// ---- 20_Product/10_BCF/11_Conv/15_Subsystem/01_DUTs/ST_SubSystemData.TcDUT
TYPE ST_SubsystemData :
(**************************************************************************************
 * 	Application		:	BoxControl Framework
 *	Revision		:	$Revision: 404529 $
 *	Revision date	:	$Date: 2018-04-23 08:21:38 +0200 (Mo., 23 Apr 2018) $
 *	Last changed by	:	$Author: b7bolm $
 *	URL				:	$URL: http://almscdc.swisslog.com/repo/SWPD/Development/BoxControlFramework/20_Release/trunk/01_Software/BCF/BCF/JumpStart/20_Product/10_App/15_Subsystem/10_Lib/10_Conv/01_DUTs/ST_SubSystemData.TcDUT $
 *
 *	Purpose			:	Subsystem data
 *
 * ------------------------------------------------------------------------------------
 *	Copyright Swisslog [IP AG], Switzerland. All rights reserved.
 * 
 * ------------------------------------------------------------------------------------
 *	
 * 	Revision History: 
 *
 * 	VERSION			DATE			INITIALS			DESCRIPTION
 *	0.1				01.01.2001		swl					Example
 *
 **************************************************************************************)
STRUCT
	Init			: BOOL; // Initialized
	InitRunning		: BOOL; // Init ongoing
	OperationState	: ST_PositionState; // Subsystem state
	ErrorData		: ST_SubsystemErrorStruct; // Error data set 
END_STRUCT
END_TYPE

// ---- 20_Product/10_BCF/11_Conv/15_Subsystem/01_DUTs/ST_SubSystemErrorStruct.TcDUT
TYPE ST_SubsystemErrorStruct :
(**************************************************************************************
 * 	Application		:	BoxControl Framework
 *	Revision		:	$Revision: 404529 $
 *	Revision date	:	$Date: 2018-04-23 08:21:38 +0200 (Mo., 23 Apr 2018) $
 *	Last changed by	:	$Author: b7bolm $
 *	URL				:	$URL: http://almscdc.swisslog.com/repo/SWPD/Development/BoxControlFramework/20_Release/trunk/01_Software/BCF/BCF/JumpStart/20_Product/10_App/15_Subsystem/10_Lib/10_Conv/01_DUTs/ST_SubSystemErrorStruct.TcDUT $
 *
 *	Purpose			:	Group error structure - Contains all information for the
 *						error handling.
 *
 * ------------------------------------------------------------------------------------
 *	Copyright Swisslog [IP AG], Switzerland. All rights reserved.
 * 
 * ------------------------------------------------------------------------------------
 *	
 * 	Revision History: 
 *
 * 	VERSION			DATE			INITIALS			DESCRIPTION
 *	0.1				01.01.2001		swl					Example
 *
 **************************************************************************************)
STRUCT
	ErrorState				: E_ErrorState; // Ongoing module error state
	Error					: ST_ErrorDataSet; // Ongoing reported error
	DataSetIdx				: INT; // Choosen error set index
	ErrorDataSet			: ARRAY [1..NUMBER_OF_ERROR_SETS] OF ST_ErrorDataSet; // Overview about all message sets
	ExternalError			: ST_ErrorDataSet; // External error, Can be set customized or by control code
	GroupErrorPending		: BOOL; // A group is in error state
END_STRUCT
END_TYPE

// ---- 20_Product/10_BCF/11_Conv/15_Subsystem/01_DUTs/ST_SubSystemInterface.TcDUT
TYPE ST_SubsystemInterface :
(**************************************************************************************
 * 	Application		:	BoxControl Framework
 *	Revision		:	$Revision: 404529 $
 *	Revision date	:	$Date: 2018-04-23 08:21:38 +0200 (Mo., 23 Apr 2018) $
 *	Last changed by	:	$Author: b7bolm $
 *	URL				:	$URL: http://almscdc.swisslog.com/repo/SWPD/Development/BoxControlFramework/20_Release/trunk/01_Software/BCF/BCF/JumpStart/20_Product/10_App/15_Subsystem/10_Lib/10_Conv/01_DUTs/ST_SubSystemInterface.TcDUT $
 *
 *	Purpose			:	
 *
 * ------------------------------------------------------------------------------------
 *	Copyright Swisslog [IP AG], Switzerland. All rights reserved.
 * 
 * ------------------------------------------------------------------------------------
 *	
 * 	Revision History: 
 *
 * 	VERSION			DATE			INITIALS			DESCRIPTION
 *	0.1				01.01.2001		swl					Example
 *
 **************************************************************************************)
STRUCT
	In			: ST_SubSystemInterfaceIn;
	Out			: ST_SubSystemInterfaceOut;
END_STRUCT
END_TYPE

// ---- 20_Product/10_BCF/11_Conv/15_Subsystem/01_DUTs/ST_SubSystemInterfaceIn.TcDUT
TYPE ST_SubSystemInterfaceIn :
(**************************************************************************************
 * 	Application		:	BoxControl Framework
 *	Revision		:	$Revision: 404529 $
 *	Revision date	:	$Date: 2018-04-23 08:21:38 +0200 (Mo., 23 Apr 2018) $
 *	Last changed by	:	$Author: b7bolm $
 *	URL				:	$URL: http://almscdc.swisslog.com/repo/SWPD/Development/BoxControlFramework/20_Release/trunk/01_Software/BCF/BCF/JumpStart/20_Product/10_App/15_Subsystem/10_Lib/10_Conv/01_DUTs/ST_SubSystemInterfaceIn.TcDUT $
 *
 *	Purpose			:	
 *
 * ------------------------------------------------------------------------------------
 *	Copyright Swisslog [IP AG], Switzerland. All rights reserved.
 * 
 * ------------------------------------------------------------------------------------
 *	
 * 	Revision History: 
 *
 * 	VERSION			DATE			INITIALS			DESCRIPTION
 *	0.1				01.01.2001		swl					Example
 *
 **************************************************************************************)
STRUCT
	MasterSpeed					: INT; // Incoming Master speed request
END_STRUCT
END_TYPE

// ---- 20_Product/10_BCF/11_Conv/15_Subsystem/01_DUTs/ST_SubSystemInterfaceOut.TcDUT
TYPE ST_SubSystemInterfaceOut :
(**************************************************************************************
 * 	Application		:	BoxControl Framework
 *	Revision		:	$Revision: 404529 $
 *	Revision date	:	$Date: 2018-04-23 08:21:38 +0200 (Mo., 23 Apr 2018) $
 *	Last changed by	:	$Author: b7bolm $
 *	URL				:	$URL: http://almscdc.swisslog.com/repo/SWPD/Development/BoxControlFramework/20_Release/trunk/01_Software/BCF/BCF/JumpStart/20_Product/10_App/15_Subsystem/10_Lib/10_Conv/01_DUTs/ST_SubSystemInterfaceOut.TcDUT $
 *
 *	Purpose			:	
 *
 * ------------------------------------------------------------------------------------
 *	Copyright Swisslog [IP AG], Switzerland. All rights reserved.
 * 
 * ------------------------------------------------------------------------------------
 *	
 * 	Revision History: 
 *
 * 	VERSION			DATE			INITIALS			DESCRIPTION
 *	0.1				01.01.2001		swl					Example
 *
 **************************************************************************************)
STRUCT
	MasterSpeed					: INT; // Valid master speed
END_STRUCT
END_TYPE

// ---- 20_Product/20_ProBox/10_Base/01_DUTs/E_ErrorProduct.TcDUT
{attribute 'qualified_only'}
{attribute 'strict'}
(**************************************************************************************
 * 	Application		:	BoxControl Framework
 *	Revision		:	$Revision: 417092 $
 *	Revision date	:	$Date: 2018-11-14 12:58:58 +0100 (Mi., 14 Nov 2018) $
 *	Last changed by	:	$Author: q8aberh $
 *	URL				:	$URL: http://almscdc.swisslog.com/repo/SWPD/Development/ProMove/02_Controls/ProBox/03_Implementation/01_DevelopmentProject/01_Software/ProBox_COE/ProBox_DevProj_v1.0/PLC_1/20_Product/10_App/10_Base/E_ErrorProduct.TcDUT $
 *
 *	Purpose			:	Product error
 *						This Structure can be used for product specific error codes.
 *						ATTENTION! - WM needs to be updated for each error code
 *
 *						0 - 999 Reserved Framework
 *						1000... Product specific
 *
 * ------------------------------------------------------------------------------------
 *	Copyright Swisslog [IP AG], Switzerland. All rights reserved.
 * 
 * ------------------------------------------------------------------------------------
 *	
 * 	Revision History: 
 *
 * 	VERSION			DATE			INITIALS			DESCRIPTION
 *	0.1				01.01.2001		swl					Example
 *
 **************************************************************************************)
TYPE E_ErrorProduct :
(
	UNDEF := 1000,	
(* -------------------------------------------------------------
		ProBox error messages
--------------------------------------------------------------*)
	SCALE_OVER_UNDER_WEIGHT							:= 1100,
	SCALE_WEIGHT_CELL_ERROR							:= 1101
	
);
END_TYPE

// ---- 20_Product/20_ProBox/22_ProMove/01_DUTs/ASI/ST_ASI_HW_Input.TcDUT
TYPE ST_ASI_HW_Input :
STRUCT
	A_1_15              AT %I* : ST_HW_InputsASi_1_15;  //Slave A 1..15
	A_16_31             AT %I* : ST_HW_InputsASi_16_31; //Slave A 16..31
	B_1_15              AT %I* : ST_HW_InputsASi_1_15;  //Slave B 1..15
	B_16_31             AT %I* : ST_HW_InputsASi_16_31; //Slave B 16..31
END_STRUCT
END_TYPE

// ---- 20_Product/20_ProBox/22_ProMove/01_DUTs/ASI/ST_ASI_HW_IO.TcDUT
TYPE ST_ASI_HW_IO :
STRUCT
	I 	AT %I* : ST_ASI_HW_Input; //ASI Ring 1 Inputs
	//I2 : ST_ASI_HW_Input; //ASI Ring 2 Inputs
	Q 	AT %Q* : ST_ASI_HW_Output; //ASI ring 1 Outputs
	//Q2 : ST_ASI_HW_Output; //ASI ring 2 Outputs
END_STRUCT
END_TYPE

// ---- 20_Product/20_ProBox/22_ProMove/01_DUTs/ASI/ST_ASI_HW_Output.TcDUT
TYPE ST_ASI_HW_Output :
STRUCT
	A_1_15              AT %Q* : ST_HW_OutputsASi_1_15;  //Slave A 1..15
	A_16_31             AT %Q* : ST_HW_OutputsASi_16_31; //Slave A 16..31
	B_1_15              AT %Q* : ST_HW_OutputsASi_1_15;  //Slave B 1..15
	B_16_31             AT %Q* : ST_HW_OutputsASi_16_31; //Slave B 16..31
END_STRUCT
END_TYPE

// ---- 20_Product/20_ProBox/22_ProMove/01_DUTs/ASI/ST_HW_InputsASi_16_31.TcDUT
TYPE ST_HW_InputsASi_16_31 :
STRUCT
	IN_17_1	: BIT;
	IN_17_2	: BIT;
	IN_17_3	: BIT;
	IN_17_4 	: BIT;
	
	IN_16_1	: BIT;
	IN_16_2	: BIT;
	IN_16_3	: BIT;
	IN_16_4 	: BIT;

	IN_19_1	: BIT;
	IN_19_2	: BIT;
	IN_19_3	: BIT;
	IN_19_4	: BIT;

	IN_18_1	: BIT;
	IN_18_2	: BIT;
	IN_18_3	: BIT;
	IN_18_4	: BIT;

	IN_21_1	: BIT;
	IN_21_2	: BIT;
	IN_21_3	: BIT;
	IN_21_4 	: BIT;
	
	IN_20_1	: BIT;
	IN_20_2	: BIT;
	IN_20_3	: BIT;
	IN_20_4	: BIT;

	IN_23_1	: BIT;
	IN_23_2	: BIT;
	IN_23_3	: BIT;
	IN_23_4 	: BIT;

	IN_22_1	: BIT;
	IN_22_2	: BIT;
	IN_22_3	: BIT;
	IN_22_4	: BIT;

	IN_25_1	: BIT;
	IN_25_2	: BIT;
	IN_25_3	: BIT;
	IN_25_4	: BIT;

	IN_24_1	: BIT;
	IN_24_2	: BIT;
	IN_24_3	: BIT;
	IN_24_4	: BIT;

	IN_27_1	: BIT;
	IN_27_2	: BIT;
	IN_27_3	: BIT;
	IN_27_4	: BIT;

	IN_26_1	: BIT;
	IN_26_2	: BIT;
	IN_26_3	: BIT;
	IN_26_4	: BIT;

	IN_29_1	: BIT;
	IN_29_2	: BIT;
	IN_29_3	: BIT;
	IN_29_4	: BIT;

	IN_28_1	: BIT;
	IN_28_2	: BIT;
	IN_28_3	: BIT;
	IN_28_4	: BIT;
	
	IN_31_1	: BIT;
	IN_31_2	: BIT;
	IN_31_3	: BIT;
	IN_31_4	: BIT;

	IN_30_1	: BIT;
	IN_30_2	: BIT;
	IN_30_3	: BIT;
	IN_30_4	: BIT;
END_STRUCT
END_TYPE

// ---- 20_Product/20_ProBox/22_ProMove/01_DUTs/ASI/ST_HW_InputsASi_1_15.TcDUT
TYPE ST_HW_InputsASi_1_15 :
STRUCT
	IN_1_1	: BIT;
	IN_1_2	: BIT;
	IN_1_3	: BIT;
	IN_1_4 	: BIT;
	
	CONF_ERR		: BIT;
	ASI_POWER_FAULT	: BIT;
	NODE_ERROR		: BIT;
	CONFIG_MODE		: BIT;

	IN_3_1	: BIT;
	IN_3_2	: BIT;
	IN_3_3	: BIT;
	IN_3_4 	: BIT;

	IN_2_1	: BIT;
	IN_2_2	: BIT;
	IN_2_3	: BIT;
	IN_2_4 	: BIT;

	IN_5_1	: BIT;
	IN_5_2	: BIT;
	IN_5_3	: BIT;
	IN_5_4 	: BIT;
	
	IN_4_1	: BIT;
	IN_4_2	: BIT;
	IN_4_3	: BIT;
	IN_4_4 	: BIT;

	IN_7_1	: BIT;
	IN_7_2	: BIT;
	IN_7_3	: BIT;
	IN_7_4 	: BIT;

	IN_6_1	: BIT;
	IN_6_2	: BIT;
	IN_6_3	: BIT;
	IN_6_4 	: BIT;

	IN_9_1	: BIT;
	IN_9_2	: BIT;
	IN_9_3	: BIT;
	IN_9_4 	: BIT;

	IN_8_1	: BIT;
	IN_8_2	: BIT;
	IN_8_3	: BIT;
	IN_8_4 	: BIT;

	IN_11_1	: BIT;
	IN_11_2	: BIT;
	IN_11_3	: BIT;
	IN_11_4	: BIT;

	IN_10_1	: BIT;
	IN_10_2	: BIT;
	IN_10_3	: BIT;
	IN_10_4	: BIT;

	IN_13_1	: BIT;
	IN_13_2	: BIT;
	IN_13_3	: BIT;
	IN_13_4	: BIT;

	IN_12_1	: BIT;
	IN_12_2	: BIT;
	IN_12_3	: BIT;
	IN_12_4	: BIT;
	
	IN_15_1	: BIT;
	IN_15_2	: BIT;
	IN_15_3	: BIT;
	IN_15_4	: BIT;

	IN_14_1	: BIT;
	IN_14_2	: BIT;
	IN_14_3	: BIT;
	IN_14_4	: BIT;
END_STRUCT
END_TYPE

// ---- 20_Product/20_ProBox/22_ProMove/01_DUTs/ASI/ST_HW_OutputsASi_16_31.TcDUT
TYPE ST_HW_OutputsASi_16_31 :
STRUCT
	OUT_17_1	: BIT;
	OUT_17_2	: BIT;
	OUT_17_3	: BIT;
	OUT_17_4 	: BIT;
	
	OUT_16_1	: BIT;
	OUT_16_2	: BIT;
	OUT_16_3	: BIT;
	OUT_16_4 	: BIT;

	OUT_19_1	: BIT;
	OUT_19_2	: BIT;
	OUT_19_3	: BIT;
	OUT_19_4	: BIT;

	OUT_18_1	: BIT;
	OUT_18_2	: BIT;
	OUT_18_3	: BIT;
	OUT_18_4	: BIT;

	OUT_21_1	: BIT;
	OUT_21_2	: BIT;
	OUT_21_3	: BIT;
	OUT_21_4 	: BIT;
	
	OUT_20_1	: BIT;
	OUT_20_2	: BIT;
	OUT_20_3	: BIT;
	OUT_20_4	: BIT;

	OUT_23_1	: BIT;
	OUT_23_2	: BIT;
	OUT_23_3	: BIT;
	OUT_23_4 	: BIT;

	OUT_22_1	: BIT;
	OUT_22_2	: BIT;
	OUT_22_3	: BIT;
	OUT_22_4	: BIT;

	OUT_25_1	: BIT;
	OUT_25_2	: BIT;
	OUT_25_3	: BIT;
	OUT_25_4	: BIT;

	OUT_24_1	: BIT;
	OUT_24_2	: BIT;
	OUT_24_3	: BIT;
	OUT_24_4	: BIT;

	OUT_27_1	: BIT;
	OUT_27_2	: BIT;
	OUT_27_3	: BIT;
	OUT_27_4	: BIT;

	OUT_26_1	: BIT;
	OUT_26_2	: BIT;
	OUT_26_3	: BIT;
	OUT_26_4	: BIT;

	OUT_29_1	: BIT;
	OUT_29_2	: BIT;
	OUT_29_3	: BIT;
	OUT_29_4	: BIT;

	OUT_28_1	: BIT;
	OUT_28_2	: BIT;
	OUT_28_3	: BIT;
	OUT_28_4	: BIT;
	
	OUT_31_1	: BIT;
	OUT_31_2	: BIT;
	OUT_31_3	: BIT;
	OUT_31_4	: BIT;

	OUT_30_1	: BIT;
	OUT_30_2	: BIT;
	OUT_30_3	: BIT;
	OUT_30_4	: BIT;
END_STRUCT
END_TYPE

// ---- 20_Product/20_ProBox/22_ProMove/01_DUTs/ASI/ST_HW_OutputsASi_1_15.TcDUT
TYPE ST_HW_OutputsASi_1_15 :
STRUCT
	OUT_1_1	: BIT;
	OUT_1_2	: BIT;
	OUT_1_3	: BIT;
	OUT_1_4 : BIT;
	
	SET_OFFLINE			: BIT;
	LOS_MASTER_BIT		: BIT;
	SET_CONFIG_MODE		: BIT;
	SET_PROTECTED_MODE	: BIT;

	OUT_3_1	: BIT;
	OUT_3_2	: BIT;
	OUT_3_3	: BIT;
	OUT_3_4 : BIT;

	OUT_2_1	: BIT;
	OUT_2_2	: BIT;
	OUT_2_3	: BIT;
	OUT_2_4 : BIT;

	OUT_5_1	: BIT;
	OUT_5_2	: BIT;
	OUT_5_3	: BIT;
	OUT_5_4 : BIT;
	
	OUT_4_1	: BIT;
	OUT_4_2	: BIT;
	OUT_4_3	: BIT;
	OUT_4_4 : BIT;

	OUT_7_1	: BIT;
	OUT_7_2	: BIT;
	OUT_7_3	: BIT;
	OUT_7_4 : BIT;

	OUT_6_1	: BIT;
	OUT_6_2	: BIT;
	OUT_6_3	: BIT;
	OUT_6_4 : BIT;

	OUT_9_1	: BIT;
	OUT_9_2	: BIT;
	OUT_9_3	: BIT;
	OUT_9_4 : BIT;

	OUT_8_1	: BIT;
	OUT_8_2	: BIT;
	OUT_8_3	: BIT;
	OUT_8_4 : BIT;

	OUT_11_1	: BIT;
	OUT_11_2	: BIT;
	OUT_11_3	: BIT;
	OUT_11_4	: BIT;

	OUT_10_1	: BIT;
	OUT_10_2	: BIT;
	OUT_10_3	: BIT;
	OUT_10_4	: BIT;

	OUT_13_1	: BIT;
	OUT_13_2	: BIT;
	OUT_13_3	: BIT;
	OUT_13_4	: BIT;

	OUT_12_1	: BIT;
	OUT_12_2	: BIT;
	OUT_12_3	: BIT;
	OUT_12_4	: BIT;
	
	OUT_15_1	: BIT;
	OUT_15_2	: BIT;
	OUT_15_3	: BIT;
	OUT_15_4	: BIT;

	OUT_14_1	: BIT;
	OUT_14_2	: BIT;
	OUT_14_3	: BIT;
	OUT_14_4	: BIT;
END_STRUCT
END_TYPE

// ---- 20_Product/20_ProBox/22_ProMove/01_DUTs/E_Axis_Orientation.TcDUT
TYPE E_Axis_Orientation :
(**************************************************************************************
 * 	Application		:	BoxControl Framework
 *	Revision		:	$Revision: 417092 $
 *	Revision date	:	$Date: 2018-11-14 12:58:58 +0100 (Mi., 14 Nov 2018) $
 *	Last changed by	:	$Author: q8aberh $
 *	URL				:	$URL: http://almscdc.swisslog.com/repo/SWPD/Development/ProMove/02_Controls/ProBox/03_Implementation/01_DevelopmentProject/01_Software/ProBox_COE/ProBox_DevProj_v1.0/PLC_1/20_Product/10_App/12_E_Functions/11_ProBox/01_DUTs/E_Axis_Orientation.TcDUT $
 *
 *	Purpose			:	orientation of function axis on element 
 *
 * ------------------------------------------------------------------------------------
 *	Copyright Swisslog [IP AG], Switzerland. All rights reserved.
 * 
 * ------------------------------------------------------------------------------------
 *	
 * 	Revision History: 
 *
 * 	VERSION			DATE			INITIALS			DESCRIPTION
 *	0.1				15.06.2018		lca					Example
 *
 **************************************************************************************)	
(
	IDLE, // Funciton axis is not requested by an element
	Element_12, // Funciton axis is requested by the element axis 1-2 in the same direction
	Element_21, // Funciton axis is requested by the element axis 1-2 in the opposite direction
	Element_34, // Funciton axis is requested by the element axis 3-4 in the same direction
	Element_43  // Funciton axis is requested by the element axis 3-4 in the opposite direction	
);
END_TYPE

// ---- 20_Product/20_ProBox/22_ProMove/01_DUTs/E_ProBoxMotorSpeed.TcDUT
TYPE E_ProBoxMotorSpeed :
(**************************************************************************************
 * 	Application		:	BoxControl Framework
 *	Revision		:	$Revision: 418851 $
 *	Revision date	:	$Date: 2018-12-11 17:28:45 +0100 (Di., 11 Dez 2018) $
 *	Last changed by	:	$Author: Q8OTTOC $
 *	URL				:	$URL: http://almscdc.swisslog.com/repo/SWPD/Development/ProMove/02_Controls/ProBox/03_Implementation/01_DevelopmentProject/01_Software/ProBox_COE/ProBox_DevProj_v1.0/PLC_1/20_Product/10_App/12_E_Functions/11_ProBox/01_DUTs/E_ProBoxMotorSpeed.TcDUT $
 *
 *	Purpose			:	Motor speed
 *
 * ------------------------------------------------------------------------------------
 *	Copyright Swisslog [IP AG], Switzerland. All rights reserved.
 * 
 * ------------------------------------------------------------------------------------
 *	
 * 	Revision History: 
 *
 * 	VERSION			DATE			INITIALS			DESCRIPTION
 *	0.1				13.04.2018		PkF					First version of motor speeds
  *	0.2				29.11.2018		lca					Sorted from lowest to highest speed
 *
 **************************************************************************************)
(
	CREEP_SPEED,
	LOW_SPEED,
	NORMAL	
);
END_TYPE

// ---- 20_Product/20_ProBox/22_ProMove/15_SubSystem/01_DUTs/ST_CFG_ProBoxSubsystem.TcDUT
TYPE ST_CFG_ProBoxSubsystem :
STRUCT
	AM_Exists					: BOOL; // Automation manager is existing
	SPOC_Exists					: BOOL; // SPOC exists			
	tRequestReset				: TIME; // Time to reset a request
	tDelayMonitoring			: TIME; // Time to delay monitoring	
	tDelayStopping				: TIME; // Time to delay stopping
	EnableTimeSync				: BOOL; // Enable time sync
	MinTimeSync					: TIME; // Minimal time sync value
	CPU_FanExists				: BOOL; // Is true if CPU with fan equiped 
	MinFanSpeed					: UINT; // Min FAN speed
	CPU_UsageWarning			: INT; // CPU usage warning [%]
	CPU_UsageError				: INT; // CPU usage error [%]
	CPU_TemperatureWarning		: INT; // CPU temperatur warning
	CPU_TemperatureError		: INT; // CPU temperatur error
END_STRUCT
END_TYPE

// ---- 20_Product/20_ProBox/30_Toolbox/12_DUTs/E_PalletOrientation.TcDUT
TYPE E_PalletOrientation :
(
	OrientationZero,
	OrientationNinty,
	OrientationOneEighty,
	OrientationTwoSeventy
);
END_TYPE

// ---- 20_Product/20_ProBox/30_Toolbox/70_Strategies/01_DUTs/ST_FifoBuffer.TcDUT
TYPE ST_FifoBuffer :
STRUCT
	Occupied 			: BOOL;
	EntryOK 			: BOOL;
	eFunctionNumber		: E_FunctionNumber;
	Priority 			: INT;
	//TU_Indexs			: ARRAY [1..NUMBER_OF_ZONES_PER_FUNCTION] OF DINT;  //store the TU index for all zones	
END_STRUCT
END_TYPE

// ---- 20_Product/20_ProBox/30_Toolbox/70_Strategies/01_DUTs/ST_RoutingSluggingData.TcDUT
TYPE ST_RoutingSluggingData :
STRUCT
	FunctionsBehind 		: ARRAY[1..20] OF E_FunctionNumber; // Functions to check before function (back)
	FunctionsInfront		: ARRAY[1..20] OF E_FunctionNumber; // Functions to check after function (forward)
	InvalidDestinations		: ARRAY[1..20] OF E_FunctionNumber; // Destinations of pallets behind that should not be considered slugging with
END_STRUCT
END_TYPE

// ---- 20_Product/20_ProBox/40_TC_Visualization/15_PowerStore/DTUs/ST_AccessPanel.TcDUT
TYPE ST_AccessPanel :
STRUCT
	inputs : ST_AccessPanelInputs;
	outputs : ST_AccessPanelOutputs;
END_STRUCT
END_TYPE

// ---- 20_Product/20_ProBox/40_TC_Visualization/15_PowerStore/DTUs/ST_AccessPanelInputs.TcDUT
TYPE ST_AccessPanelInputs :
STRUCT
	PB_ActivateMainContactor : BOOL; // Pushbutton activate main contactor
	PB_AutoOn : BOOL; // Pushbutton activate automatic mode
	PB_EmergencyStopReset : BOOL; // Pushbutton reset emergency stop
	PB_ErrorReset : BOOL; // Pushbutton reset error
	PB_EmergencyStop : BOOL; // Pushbutton Emergency stop
	SW_EntryRequest : BOOL; // Auto/Entry request switch
END_STRUCT
END_TYPE

// ---- 20_Product/20_ProBox/40_TC_Visualization/15_PowerStore/DTUs/ST_AccessPanelOutputs.TcDUT
TYPE ST_AccessPanelOutputs :
STRUCT
	LED_MainContactorActivated :BOOL; // LED-lamp main contactor is activated
	LED_AutoIsOn : BOOL; // LED-lamp automatic mode is activated
	LED_ClearEnterance : BOOL; // LED-lamp clear to enter
	LED_EmergencyStop : BOOL; // LED-lamp emergency stop
	LED_Error : BOOL; // LED-lamp error
END_STRUCT
END_TYPE

// ---- 20_Product/20_ProBox/40_TC_Visualization/15_PowerStore/DTUs/ST_AKcabinetPanel.TcDUT
TYPE ST_AKcabinetPanel :
STRUCT
	inputs : ST_AKcabinetPanelInputs;
	outputs : ST_AKcabinetPanelOutputs;
END_STRUCT
END_TYPE

// ---- 20_Product/20_ProBox/40_TC_Visualization/15_PowerStore/DTUs/ST_AKcabinetPanelInputs.TcDUT
TYPE ST_AKcabinetPanelInputs :
STRUCT
	PB_ActivateMainContactor : BOOL; // Pushbutton activate main contactor
	PB_MainContactorOff : BOOL; // Pushbutton main contactor off
	PB_AutoOn : BOOL; // Pushbutton activate automatic mode
	PB_EmergencyStopReset : BOOL; // Pushbutton reset emergency stop
	PB_ErrorReset : BOOL; // Pushbutton reset error
	PB_EmergencyStop : BOOL; // Pushbutton Emergency stop
	SW_Auto : BOOL; // Auto/Man keyswitch
	PB_VcUp : BOOL; // Lift up vertical conveyor
	PB_VcDown : BOOL; // Lift down vertical conveyor
	
	PB_VcConvLeft : BOOL; // Vertical conveyor Left
	PB_VcConvRight : BOOL; // Vertical conveyor Right
 	
	SW_EntryRequest : BOOL; // Auto/Entry request switch
	SW_EmergencyDrive : BOOL; // Emergency drive
	
END_STRUCT
END_TYPE

// ---- 20_Product/20_ProBox/40_TC_Visualization/15_PowerStore/DTUs/ST_AKcabinetPanelOutputs.TcDUT
TYPE ST_AKcabinetPanelOutputs :
STRUCT
	LED_MainContactorActivated :BOOL; // LED-lamp main contactor is activated
	LED_AutoIsOn : BOOL; // LED-lamp automatic mode is activated
	LED_ClearEnterance : BOOL; // LED-lamp clear to enter
	LED_EmergencyStop : BOOL; // LED-lamp emergency stop
	LED_Error : BOOL; // LED-lamp error
END_STRUCT
END_TYPE

// ---- 20_Product/20_ProBox/40_TC_Visualization/15_PowerStore/DTUs/ST_TransferPanel.TcDUT
TYPE ST_TransferPanel :
STRUCT
	inputs : ST_TransferPanelInputs;
	outputs : ST_TransferPanelOutputs;
END_STRUCT
END_TYPE

// ---- 20_Product/20_ProBox/40_TC_Visualization/15_PowerStore/DTUs/ST_TransferPanelInputs.TcDUT
TYPE ST_TransferPanelInputs :
STRUCT
	PB_ActivateMainContactor : BOOL; // Pushbutton activate main contactor
	PB_MainContactorOff : BOOL; // Pushbutton main contactor off
	PB_AutoOn : BOOL; // Pushbutton activate automatic mode
	PB_EmergencyStopReset : BOOL; // Pushbutton reset emergency stop
	PB_ErrorReset : BOOL; // Pushbutton reset error
	PB_EmergencyStop : BOOL; // Pushbutton Emergency stop
	SW_Auto : BOOL; // Auto/Man keyswitch
	PB_VcUp : BOOL; // Lift up vertical conveyor
	PB_VcDown : BOOL; // Lift down vertical conveyor
	
	PB_VcConvLeft : BOOL; // Vertical conveyor Left
	PB_VcConvRight : BOOL; // Vertical conveyor Right
 	PB_Conv_1_Left : BOOL; // Conveyor 1 Left
	PB_Conv_1_Right : BOOL; // Conveyor 1 Right
	PB_Conv_2_Left : BOOL; // Conveyor 2 Left
	PB_Conv_2_Right : BOOL; // Conveyor 2 Right
	PB_Conv_3_Left : BOOL; // Conveyor 3 Left
	PB_Conv_3_Right : BOOL; // Conveyor 3 Right
	
	PB_AC_ConvLeft : BOOL; // Aisle carrier conveyor Left
	PB_AC_ConvRight : BOOL; // Aisle carrier conveyor Right
	
END_STRUCT
END_TYPE

// ---- 20_Product/20_ProBox/40_TC_Visualization/15_PowerStore/DTUs/ST_TransferPanelOutputs.TcDUT
TYPE ST_TransferPanelOutputs :
STRUCT
	LED_MainContactorActivated :BOOL; // LED-lamp main contactor is activated
	LED_AutoIsOn : BOOL; // LED-lamp automatic mode is activated
	LED_VcStopped : BOOL; // LED-lamp vertical conveyor stopped
	LED_EmergencyStop : BOOL; // LED-lamp emergency stop
	LED_Error : BOOL; // LED-lamp error
END_STRUCT
END_TYPE

// ---- 20_Product/20_ProBox/40_TC_Visualization/15_PowerStore/DTUs/ST_VC_AccessPanel.TcDUT
TYPE ST_VC_AccessPanel :
STRUCT
	inputs : ST_VC_AccessPanelInputs;
	outputs : ST_VC_AccessPanelOutputs;
END_STRUCT
END_TYPE

// ---- 20_Product/20_ProBox/40_TC_Visualization/15_PowerStore/DTUs/ST_VC_AccessPanelInputs.TcDUT
TYPE ST_VC_AccessPanelInputs :
STRUCT
	PB_ActivateMainContactor : BOOL; // Pushbutton activate main contactor
	PB_MainContactorOff : BOOL; // Pushbutton main contactor off
	PB_AutoOn : BOOL; // Pushbutton activate automatic mode
	PB_EmergencyStopReset : BOOL; // Pushbutton reset emergency stop
	PB_ErrorReset : BOOL; // Pushbutton reset error
	PB_EmergencyStop : BOOL; // Pushbutton Emergency stop
	SW_Auto : BOOL; // Auto/Man keyswitch
	PB_VcUp : BOOL; // Lift up vertical conveyor
	PB_VcDown : BOOL; // Lift down vertical conveyor
	
	PB_VcConvLeft : BOOL; // Vertical conveyor Left
	PB_VcConvRight : BOOL; // Vertical conveyor Right
 	
	SW_EntryRequest : BOOL; // Auto/Entry request switch
	SW_EmergencyDrive : BOOL; // Emergency drive
	
END_STRUCT
END_TYPE

// ---- 20_Product/20_ProBox/40_TC_Visualization/15_PowerStore/DTUs/ST_VC_AccessPanelOutputs.TcDUT
TYPE ST_VC_AccessPanelOutputs :
STRUCT
	LED_MainContactorActivated :BOOL; // LED-lamp main contactor is activated
	LED_AutoIsOn : BOOL; // LED-lamp automatic mode is activated
	LED_ClearEnterance : BOOL; // LED-lamp clear to enter
	LED_EmergencyStop : BOOL; // LED-lamp emergency stop
	LED_Error : BOOL; // LED-lamp error
END_STRUCT
END_TYPE

// ---- 20_Product/30_Toolbox/11_Com/10_TCP_Driver/01_DUTs/E_ConnStates.TcDUT
TYPE E_ConnStates :
(**************************************************************************************
 * 	AUTHOR		Swisslog
 * 	LIBRARY		Data types/02_Library/02_Communication/TCP-Driver
 *	RELEASE		1.0.0
 * ------------------------------------------------------------------------------------
 * 	Revision History: 
 *
 * 	VERSION		DATE		INITIALS	DESCRIPTION
 *	0.1		07.09.2011	swl		initial version
 **************************************************************************************)
(
	CONN_IDLE,  // 0
	CONN_RUNNING, // 1
	CONN_CLOSE, // 2
	CONN_ERROR // 3
);
END_TYPE

// ---- 20_Product/30_Toolbox/11_Com/10_TCP_Driver/01_DUTs/E_RecvStates.TcDUT
TYPE E_RecvStates :
(**************************************************************************************
 * 	AUTHOR		Swisslog
 * 	LIBRARY		Data types/02_Library/02_Communication/TCP-Driver
 *	RELEASE		1.0.0
 * ------------------------------------------------------------------------------------
 * 	Revision History: 
 *
 * 	VERSION		DATE		INITIALS	DESCRIPTION
 *	0.1		07.09.2011	swl		initial version
 **************************************************************************************)
(
	RECV_IDLE,
	RECV_WAIT,
	RECV_ERROR
);
END_TYPE

// ---- 20_Product/30_Toolbox/11_Com/10_TCP_Driver/01_DUTs/E_SendStates.TcDUT
TYPE E_SendStates :
(**************************************************************************************
 * 	AUTHOR		Swisslog
 * 	LIBRARY		Data types/02_Library/02_Communication/TCP-Driver
 *	RELEASE		1.0.0
 * ------------------------------------------------------------------------------------
 * 	Revision History: 
 *
 * 	VERSION		DATE		INITIALS	DESCRIPTION
 *	0.1		07.09.2011	swl		initial version
 **************************************************************************************)
(
	SEND_IDLE,
	SEND_WAIT,
	SEND_ERROR
);
END_TYPE

// ---- 20_Product/30_Toolbox/11_Com/10_TCP_Driver/01_DUTs/E_ServStates.TcDUT
TYPE E_ServStates :
(**************************************************************************************
 * 	AUTHOR		Swisslog
 * 	LIBRARY		Data types/02_Library/02_Communication/TCP-Driver
 *	RELEASE		1.0.0
 * ------------------------------------------------------------------------------------
 * 	Revision History: 
 *
 * 	VERSION		DATE		INITIALS	DESCRIPTION
 *	0.1		07.09.2011	swl		initial version
 **************************************************************************************)
(
	ACCEPT_IDLE,
	ACCEPT_OPEN_START,
	ACCEPT_OPEN_WAIT,
	CLIENT_CONNECTED,
	ACCEPT_CLOSE_START,
	ACCEPT_CLOSE_WAIT,
	ACCEPT_ERROR
);
END_TYPE

// ---- 20_Product/30_Toolbox/11_Com/10_TCP_Driver/01_DUTs/ST_CFG_TcpDriver.TcDUT
TYPE ST_CFG_TcpDriver :
(**************************************************************************************
 * 	Application		:	BoxControl Framework
 *	Revision		:	$Revision: 404529 $
 *	Revision date	:	$Date: 2018-04-23 08:21:38 +0200 (Mo., 23 Apr 2018) $
 *	Last changed by	:	$Author: b7bolm $
 *	URL				:	$URL: http://almscdc.swisslog.com/repo/SWPD/Development/BoxControlFramework/20_Release/trunk/01_Software/BCF/BCF/JumpStart/30_Toolbox/11_Com/10_TCP_Driver/01_DUTs/ST_CFG_TcpDriver.TcDUT $
 *
 *	Purpose			:	Configuration TCP/IP channel.
 *
 * ------------------------------------------------------------------------------------
 *	Copyright Swisslog [IP AG], Switzerland. All rights reserved.
 * 
 * ------------------------------------------------------------------------------------
 *	
 * 	Revision History: 
 *
 * 	VERSION			DATE			INITIALS			DESCRIPTION
 *	0.1				01.01.2001		swl					Example
 *
 **************************************************************************************)
STRUCT
	ChannelName				: STRING(80); // Name - Only for debugging
	EnableConnection		: BOOL;	// Enable channel
	RemoteHost				: STRING(15); // IP address of remote host - Client Mode Only! 
	LocalHost				: STRING(15); // IP address of local host - Server Mode Only! 
	RemotePort				: UDINT; // Port of the remote host - Client Mode Only! 
	LocalPort				: UDINT; // Port to listen on - Server Mode Only! 
	Server					: BOOL; // Is this connection to be configured as a server?  (Set to False for Client Mode) 
	ConnectTimeout			: TIME; // Timeout for connection establishment
	ClientRetryInterval		: TIME:= T#45S; // Interval for CLIENT type connections to be re-attempted - default is 45s, RetryInterval should not be lower than 30s to ensure proper execution
	ServerRetryInterval		: TIME:= T#1S; // Interval for SERVER type connections to be re-attempted - default is 1s 
	AcceptPollInterval		: TIME:= T#5S; // Interval for SERVER type connections to poll the port for incoming connection attempts - default is 5s 
	EnableDebugMsg			: BOOL; // Enables sending debug messages	
END_STRUCT
END_TYPE

// ---- 20_Product/30_Toolbox/13_TimerCounter/01_DUTs/E_PulsGen.TcDUT
TYPE E_PulsGen :
(**************************************************************************************
 * 	Application		:	BoxControl Framework
 *	Revision		:	$Revision: 404529 $
 *	Revision date	:	$Date: 2018-04-23 08:21:38 +0200 (Mo., 23 Apr 2018) $
 *	Last changed by	:	$Author: b7bolm $
 *	URL				:	$URL: http://almscdc.swisslog.com/repo/SWPD/Development/BoxControlFramework/20_Release/trunk/01_Software/BCF/BCF/JumpStart/30_Toolbox/13_TimerCounter/01_DUTs/E_PulsGen.TcDUT $
 *
 *	Purpose			:	Pulse generator
 *
 * ------------------------------------------------------------------------------------
 *	Copyright Swisslog [IP AG], Switzerland. All rights reserved.
 * 
 * ------------------------------------------------------------------------------------
 *	
 * 	Revision History: 
 *
 * 	VERSION			DATE			INITIALS			DESCRIPTION
 *	0.1				01.01.2001		swl					Example
 *
 **************************************************************************************)
(
	PG_READY,
	PG_BUSY,
	PG_END
);
END_TYPE

// ---- 20_Product/30_Toolbox/16_Sequencing/01_DUTs/ST_SeqEntry.TcDUT
/// Sequencing data set
TYPE ST_SeqEntry :
(************************************************************************************** 
* 	Application 		: BoxControl Framework 
* 	Revision 			: $Revision: 404877 $ 
* 	Revision date 		: $Date: 2018-04-26 14:10:34 +0200 (Thu, 26 Apr 2018) $ 
* 	Last changed by 	: $Author: b7ernsb $ 
* 	URL 				: $URL: http://almscdc.swisslog.com/repo/SWPD/Development/BoxControlFramework/21_Projects/BCF_2.0/trunk/BCF/BCF/JumpStart/20_Product/10_App/12_E_Functions/10_Lib/10_Conv/FB_FunctionConv.TcPOU $ 
* ------------------------------------------------------------------------------------ 
* 	© Swisslog AG 
* 	Swisslog is not liable for any usage of this source code that is not agreed 
* 	on between Swisslog and the other party. The mandatory legal liability remains 
* 	unaffected. 
* ------------------------------------------------------------------------------------ 
* 	Revision History: 
* 
* 	VERSION 		DATE 			INITIALS 			DESCRIPTION 
* 	0.1 			18.06.2018 		mbo 				Created.
* 
**************************************************************************************)
STRUCT
	TU_Index		: DINT; 
	Sequence		: ULINT; 
	SubSequence		: DINT; 
	TU_ID			: STRING(Conveyor.TU_ID_STRINGLENGTH); 
	TU_ID_HashCode	: ULINT;
	AssignmentID	: UDINT;
	Destination		: ST_PositionIdent;
	DestinationSlot : INT;
	CheckpointID	: STRING(5); 
END_STRUCT
END_TYPE

// ---- 20_Product/30_Toolbox/17_WindowTracking/10_Core/01_DUTs/E_WindowTrackingWindowState.TcDUT
/// Tracking window state
TYPE E_WindowTrackingWindowState :
(************************************************************************************** 
* 	Application 		: BoxControl Framework 
* 	Revision 			: $Revision: 408723 $ 
* 	Revision date 		: $Date: 2018-06-27 13:49:08 +0200 (Wed, 27 Jun 2018) $ 
* 	Last changed by 	: $Author: b7bolm $ 
* 	URL 				: $URL: http://almscdc.swisslog.com/repo/SWPD/Development/BoxControlFramework/21_Projects/BCF_2.0/trunk/BCF/BCF/JumpStart/20_Product/10_App/12_E_Functions/10_Lib/10_Conv/FB_FunctionList.TcPOU $ 
* ------------------------------------------------------------------------------------ 
* 	© Swisslog AG 
* 	Swisslog is not liable for any usage of this source code that is not agreed 
* 	on between Swisslog and the other party. The mandatory legal liability remains 
* 	unaffected. 
* ------------------------------------------------------------------------------------ 
* 	Revision History: 
* 
* 	VERSION 		DATE 			INITIALS 			DESCRIPTION 
* 	0.1 			24.08.2018 		ahe 				First implementation
* 
**************************************************************************************)
(
	IDLE,
	FRONT_EDGE,
	REAR_EDGE,
	OCCUPIED,
	RESERVED
);
END_TYPE

// ---- 20_Product/30_Toolbox/17_WindowTracking/10_Core/01_DUTs/ST_WindowTrackingReloc.TcDUT
TYPE ST_WindowTrackingReloc :
(************************************************************************************** 
* 	Application 		: BoxControl Framework 
* 	Revision 			: $Revision: 408723 $ 
* 	Revision date 		: $Date: 2018-06-27 13:49:08 +0200 (Wed, 27 Jun 2018) $ 
* 	Last changed by 	: $Author: b7bolm $ 
* 	URL 				: $URL: http://almscdc.swisslog.com/repo/SWPD/Development/BoxControlFramework/21_Projects/BCF_2.0/trunk/BCF/BCF/JumpStart/20_Product/10_App/12_E_Functions/10_Lib/10_Conv/FB_FunctionList.TcPOU $ 
* ------------------------------------------------------------------------------------ 
* 	© Swisslog AG 
* 	Swisslog is not liable for any usage of this source code that is not agreed 
* 	on between Swisslog and the other party. The mandatory legal liability remains 
* 	unaffected. 
* ------------------------------------------------------------------------------------ 
* 	Revision History: 
* 
* 	VERSION 		DATE 			INITIALS 			DESCRIPTION 
* 	0.1 			22.08.2018 		herzig 				First implementation
*	0.2				23.08.2018		b7bolm				Review
* 
**************************************************************************************)
STRUCT
	ZoneIndex		: UINT;
	TargetWindow 	: UINT;
END_STRUCT
END_TYPE

// ---- 20_Product/30_Toolbox/17_WindowTracking/10_Core/01_DUTs/ST_WindowTrackingTransfer.TcDUT
TYPE ST_WindowTrackingTransfer :
(**************************************************************************************
 * 	Application		:	BoxControl Framework
 *	Revision		:	$Revision: 351961 $
 *	Revision date	:	$Date: 2015-07-03 16:42:43 +0200 (Fri, 03 Jul 2015) $
 *	Last changed by	:	$Author: d7mangc $
 *	URL				:	$URL: http://almscdc.swisslog.com/repo/SWPD/Development/BoxControlFramework/20_Release/trunk/01_Software/BoxControlFramework/BoxControlFramework/JumpStart/11_Library/10_Application/10_Base/F_CompareAlphaNumericString.TcPOU $
 *
 *	Purpose			:	Window tracking trasnfer data set
 *
 * ------------------------------------------------------------------------------------
 *	Copyright Swisslog [IP AG], Switzerland. All rights reserved.
 * 
 * ------------------------------------------------------------------------------------
 *	
 * 	Revision History: 
 *
 * 	VERSION			DATE			INITIALS			DESCRIPTION
 *	0.1				01.01.2001		swl					Example 
 *
 **************************************************************************************)
STRUCT
	Active					: BOOL;
	AbsoluteInsertPosition	: UDINT;
	ZoneIndex				: UINT;
	LastWindowIndex			: UINT;
END_STRUCT
END_TYPE

// ---- 20_Product/30_Toolbox/17_WindowTracking/10_Core/01_DUTs/ST_WindowTrackingWindow.TcDUT
/// Data of one tracking window
TYPE ST_WindowTrackingWindow :
(************************************************************************************** 
* 	Application 		: BoxControl Framework 
* 	Revision 			: $Revision: 408723 $ 
* 	Revision date 		: $Date: 2018-06-27 13:49:08 +0200 (Wed, 27 Jun 2018) $ 
* 	Last changed by 	: $Author: b7bolm $ 
* 	URL 				: $URL: http://almscdc.swisslog.com/repo/SWPD/Development/BoxControlFramework/21_Projects/BCF_2.0/trunk/BCF/BCF/JumpStart/20_Product/10_App/12_E_Functions/10_Lib/10_Conv/FB_FunctionList.TcPOU $ 
* ------------------------------------------------------------------------------------ 
* 	© Swisslog AG 
* 	Swisslog is not liable for any usage of this source code that is not agreed 
* 	on between Swisslog and the other party. The mandatory legal liability remains 
* 	unaffected. 
* ------------------------------------------------------------------------------------ 
* 	Revision History: 
* 
* 	VERSION 		DATE 			INITIALS 			DESCRIPTION 
* 	0.1 			24.08.2018 		ahe 				First implementation
* 
**************************************************************************************)
STRUCT
	TU_FrontEdgePosition	: UDINT;
	TU_RearEdgePosition		: UDINT;
	State					: E_WindowTrackingWindowState;
	ZoneIndex				: UINT;
	Flush					: BOOL;
END_STRUCT
END_TYPE

// ---- 20_Product/30_Toolbox/17_WindowTracking/10_Core/01_DUTs/ST_WindowTrackingZone.TcDUT
/// Data of one tracking zone
TYPE ST_WindowTrackingZone :
(************************************************************************************** 
* 	Application 		: BoxControl Framework 
* 	Revision 			: $Revision: 408723 $ 
* 	Revision date 		: $Date: 2018-06-27 13:49:08 +0200 (Wed, 27 Jun 2018) $ 
* 	Last changed by 	: $Author: b7bolm $ 
* 	URL 				: $URL: http://almscdc.swisslog.com/repo/SWPD/Development/BoxControlFramework/21_Projects/BCF_2.0/trunk/BCF/BCF/JumpStart/20_Product/10_App/12_E_Functions/10_Lib/10_Conv/FB_FunctionList.TcPOU $ 
* ------------------------------------------------------------------------------------ 
* 	© Swisslog AG 
* 	Swisslog is not liable for any usage of this source code that is not agreed 
* 	on between Swisslog and the other party. The mandatory legal liability remains 
* 	unaffected. 
* ------------------------------------------------------------------------------------ 
* 	Revision History: 
* 
* 	VERSION 		DATE 			INITIALS 			DESCRIPTION 
* 	0.1 			24.08.2018 		ahe 				First implementation
* 
**************************************************************************************)
STRUCT
	Used					: BOOL;
	ActionId				: INT;
	ZoneLength				: UINT;
	ZoneStartWindowIndex	: UINT;
	ZoneEndWindowIndex		: UINT;
	ZoneStartPosition		: UDINT;
	ZoneEndPosition			: UDINT;
	TU_StartWindowIndex		: UINT;
	TU_EndWindowIndex		: UINT;
	TU_Present				: BOOL;
	TU_Index				: DINT;
	Flush					: BOOL; 
	InhibitShifting			: BOOL;
	PositionToLive			: UDINT;
	iActionListener			: I_TrackingActionListener;
END_STRUCT
END_TYPE

// ---- 20_Product/30_Toolbox/17_WindowTracking/10_Core/01_DUTs/ST_ZoneDataPair.TcDUT
TYPE ST_ZoneDataPair :
(************************************************************************************** 
* 	Application 		: BoxControl Framework 
* 	Revision 			: $Revision: 408723 $ 
* 	Revision date 		: $Date: 2018-06-27 13:49:08 +0200 (Wed, 27 Jun 2018) $ 
* 	Last changed by 	: $Author: b7bolm $ 
* 	URL 				: $URL: http://almscdc.swisslog.com/repo/SWPD/Development/BoxControlFramework/21_Projects/BCF_2.0/trunk/BCF/BCF/JumpStart/20_Product/10_App/12_E_Functions/10_Lib/10_Conv/FB_FunctionList.TcPOU $ 
* ------------------------------------------------------------------------------------ 
* 	© Swisslog AG 
* 	Swisslog is not liable for any usage of this source code that is not agreed 
* 	on between Swisslog and the other party. The mandatory legal liability remains 
* 	unaffected. 
* ------------------------------------------------------------------------------------ 
* 	Revision History: 
* 
* 	VERSION 		DATE 			INITIALS 			DESCRIPTION 
* 	0.1 			22.08.2018 		herzig 				First implementation
*	0.2				23.08.2018		b7bolm				Review
* 
**************************************************************************************)
STRUCT
	TrackingZoneIndex	: UINT;
	TU_Index			: DINT;
END_STRUCT
END_TYPE

// ---- 20_Product/30_Toolbox/99_Misc/01_DUTs/E_CPU_InfoStates.TcDUT
{attribute 'qualified_only'}
{attribute 'strict'}
(**************************************************************************************
 * 	Application		:	BoxControl Framework
 *	Revision		:	$Revision: 404529 $
 *	Revision date	:	$Date: 2018-04-23 08:21:38 +0200 (Mo., 23 Apr 2018) $
 *	Last changed by	:	$Author: b7bolm $
 *	URL				:	$URL: http://almscdc.swisslog.com/repo/SWPD/Development/BoxControlFramework/20_Release/trunk/01_Software/BCF/BCF/JumpStart/30_Toolbox/99_Misc/01_DUTs/E_CPU_InfoStates.TcDUT $
 *
 *	Purpose			:	Gathering CPU data
 *
 * ------------------------------------------------------------------------------------
 *	Copyright Swisslog [IP AG], Switzerland. All rights reserved.
 * 
 * ------------------------------------------------------------------------------------
 *	
 * 	Revision History: 
 *
 * 	VERSION			DATE			INITIALS			DESCRIPTION
 *	0.1				01.01.2001		swl					Example
 *
 **************************************************************************************)
TYPE E_CPU_InfoStates :
(
	INIT, 
	READ_DEVICE,
	READ_TEMPERATURE,
	READ_USAGE,
	READ_FAN,
	DONE
);
END_TYPE

// ---- 20_Product/30_Toolbox/99_Misc/13_Helper/01_DUTs/ST_TrackingZoneInfo.TcDUT
TYPE ST_TrackingZoneInfo :
(************************************************************************************** 
* 	Application 		: BoxControl Framework 
* 	Revision 			: $Revision: 408723 $ 
* 	Revision date 		: $Date: 2018-06-27 13:49:08 +0200 (Wed, 27 Jun 2018) $ 
* 	Last changed by 	: $Author: b7bolm $ 
* 	URL 				: $URL: http://almscdc.swisslog.com/repo/SWPD/Development/BoxControlFramework/21_Projects/BCF_2.0/trunk/BCF/BCF/JumpStart/20_Product/10_App/12_E_Functions/10_Lib/10_Conv/FB_FunctionList.TcPOU $ 
* ------------------------------------------------------------------------------------ 
* 	© Swisslog AG 
* 	Swisslog is not liable for any usage of this source code that is not agreed 
* 	on between Swisslog and the other party. The mandatory legal liability remains 
* 	unaffected. 
* ------------------------------------------------------------------------------------ 
* 	Revision History: 
* 
* 	VERSION 		DATE 			INITIALS 			DESCRIPTION 
* 	0.1 			30.11.2018 		mbo					First implementation
* 
**************************************************************************************)
STRUCT
	ZoneIndex		: UINT; // Tracking zone index on tracking
	PositionDelta	: DINT; // Distance to zone start. x < 0 Zone has already passed by x
	ZoneLength		: UINT; // Lengt of tracking zone
END_STRUCT
END_TYPE

// ---- 10_Project/10_App/10_Config/00_GVLs/Groups.TcGVL
///Automatically generated by BoxConfigurator 
VAR_GLOBAL
	fbSG_001                : FB_ProBOXSG;
	fbSG_002                : FB_ProBOXSG;
END_VAR

// ---- 10_Project/10_App/10_Config/00_GVLs/GVL_Safety.TcGVL
///Automatically created by BoxConfigurator
VAR_GLOBAL
END_VAR

// ---- 10_Project/10_App/10_Config/00_GVLs/HardwareMapping.TcGVL
///Automatically created by BoxConfigurator
VAR_GLOBAL
	///ASI HW I/O interface
	AK11_ASI                               : ST_ASI_HW_IO;
	///ASI HW I/O interface
	AK12_ASI                               : ST_ASI_HW_IO;
	///ASI HW I/O interface
	AK13_ASI                               : ST_ASI_HW_IO;
	///Switching group HW interface
	I_10_001_SG                     AT %I* : ST_HW_InputsSG_ProBOX;
	Q_10_001_SG                     AT %Q* : ST_HW_OutputsSG_ProBOX;
	///Switching group HW interface
	I_10_002_SG                     AT %I* : ST_HW_InputsSG_ProBOX;
	Q_10_002_SG                     AT %Q* : ST_HW_OutputsSG_ProBOX;
END_VAR

// ---- 10_Project/10_App/10_Config/00_GVLs/Positions.TcGVL
///Automatically generated by BoxConfigurator 
VAR_GLOBAL
	fbEL_10_001_0200_00_0                   : FB_ProBoxElementMotor;
	fbF_10_001_0200_01_0                    : FB_ProBoxStraightTransport;
	fbF_10_001_0200_02_0                    : FB_InOutFeedAddon;
	fbEL_10_001_0201_00_0                   : FB_ProBoxElementMotor;
	fbF_10_001_0201_01_0                    : FB_LowLiftUnit;
	fbEL_10_001_0202_00_0                   : FB_ProBoxElementMotor;
	fbF_10_001_0202_01_0                    : FB_ProBoxStraightTransport;
	fbEL_10_001_0203_00_0                   : FB_ProBoxElementMotor;
	fbF_10_001_0203_01_0                    : FB_ProBoxStraightTransport;
	fbF_10_001_0203_02_0                    : FB_ProfileCheckAddon;
	fbF_10_001_0203_03_0                    : FB_SickScannerAddon;
	fbF_10_001_0203_04_0                    : FB_TLB4WeightAddon;
	fbF_10_001_0203_05_0                    : FB_PalletCheckAddon;
	fbEL_10_001_0204_00_0                   : FB_ProBoxElementMotor;
	fbF_10_001_0204_01_0                    : FB_TurnTable;
	fbEL_10_001_0205_00_0                   : FB_ProBoxElementMotor;
	fbEL_10_001_0207_00_0                   : FB_ProBoxElementMotor;
	fbF_10_001_0207_01_0                    : FB_ProBoxStraightTransport;
	fbF_10_001_0207_02_0                    : FB_PalletMagazineAddon;
	fbEL_10_001_0208_00_0                   : FB_ProBoxElementMotor;
	fbF_10_001_0208_01_0                    : FB_ProBoxStraightTransport;
	fbEL_10_001_0209_00_0                   : FB_ProBoxElementMotor;
	fbF_10_001_0209_01_0                    : FB_TransferUnit;
	fbEL_10_001_0211_00_0                   : FB_ProBoxElementMotor;
	fbF_10_001_0211_01_0                    : FB_ProBoxStraightTransport;
	fbEL_10_001_0212_00_0                   : FB_ProBoxElementMotor;
	fbF_10_001_0212_01_0                    : FB_TransferUnit;
	fbEL_10_001_0213_00_0                   : FB_ProBoxElementMotor;
	fbF_10_001_0213_01_0                    : FB_ProBoxStraightTransport;
	fbF_10_001_0213_02_0                    : FB_PalletMagazineAddon;
	fbEL_10_001_0214_00_0                   : FB_ProBoxElementMotor;
	fbF_10_001_0214_01_0                    : FB_ProBoxStraightTransport;
	fbEL_10_001_0215_00_0                   : FB_ProBoxElementMotor;
	fbF_10_001_0215_01_0                    : FB_ProBoxStraightTransport;
	fbF_10_001_0215_02_0                    : FB_ProBoxStraightTransport;
	fbF_10_001_0215_03_0                    : FB_CraneXoverAddon;
	fbEL_10_001_0216_00_0                   : FB_ProBoxElementMotor;
	fbF_10_001_0216_01_0                    : FB_ProBoxStraightTransport;
	fbF_10_001_0216_02_0                    : FB_CraneXoverAddon;
	fbEL_10_001_0217_00_0                   : FB_ProBoxElementMotor;
	fbF_10_001_0217_01_0                    : FB_ProBoxStraightTransport;
	fbEL_10_001_0218_00_0                   : FB_ProBoxElementMotor;
	fbF_10_001_0218_01_0                    : FB_ProBoxStraightTransport;
	fbEL_10_001_0219_00_0                   : FB_ProBoxElementMotor;
	fbF_10_001_0219_01_0                    : FB_ProBoxStraightTransport;
	fbEL_10_001_0220_00_0                   : FB_ProBoxElementMotor;
	fbF_10_001_0220_01_0                    : FB_ProBoxStraightTransport;
	fbEL_10_001_0221_00_0                   : FB_ProBoxElementMotor;
	fbF_10_001_0221_01_0                    : FB_TransferUnit;
	fbEL_10_001_0222_00_0                   : FB_ProBoxElementMotor;
	fbF_10_001_0222_01_0                    : FB_TransferUnit;
	fbEL_10_001_0223_00_0                   : FB_ProBoxElementMotor;
	fbEL_10_001_0225_00_0                   : FB_ProBoxElementMotor;
	fbF_10_001_0225_01_0                    : FB_ProBoxStraightTransport;
	fbEL_10_001_0226_00_0                   : FB_ProBoxElementMotor;
	fbF_10_001_0226_01_0                    : FB_ProBoxStraightTransport;
	fbEL_10_001_0227_00_0                   : FB_ProBoxElementMotor;
	fbF_10_001_0227_01_0                    : FB_ProBoxStraightTransport;
	fbEL_10_001_0230_00_0                   : FB_ProBoxElementMotor;
	fbF_10_001_0230_01_0                    : FB_TransferCC;
	fbEL_10_001_0232_00_0                   : FB_ProBoxElementMotor;
	fbF_10_001_0232_01_0                    : FB_ProBoxStraightTransport;
	fbF_10_001_0232_02_0                    : FB_InOutFeedAddon;
	fbEL_10_001_0233_00_0                   : FB_ProBoxElementMotor;
	fbF_10_001_0233_01_0                    : FB_ProBoxStraightTransport;
	fbEL_10_002_0206_00_0                   : FB_ProBoxElementMotor;
	fbF_10_002_0206_01_0                    : FB_ProBoxStraightTransport;
END_VAR

// ---- 10_Project/10_App/10_Config/00_GVLs/ProBoxSystem.TcGVL
///Automatically created by BoxConfigurator
VAR_GLOBAL
	///Set manually to true in order to run Emulation
	EMULATION_ENABLED: BOOL:=TRUE;
	///Set manually to true in when Demo3D emulation is used.
	DEMO3D_SIM_ENABLED: BOOL:=FALSE;
	///Emulation speed. [mm/s]
	EMULATION_SPEED: INT:=1000;
	///SIS_BaseDrive - Time after a message will be repeated (Send)
	REPEAT_TIMEOUT: TIME:=T#10s;
	///SIS_BaseDrive - Time after a DUM telegram is sent
	IDLE_TIMEOUT: TIME:=T#1M;
	///SIS_BaseDrive - Time after connection will be reestablished 
	LINK_LOSS_TIMEOUT: TIME:=T#1M10s;
END_VAR

// ---- 10_Project/10_App/10_Config/00_GVLs/Subsystem.TcGVL
///Automatically created by BoxConfigurator
VAR_GLOBAL
	///Subsystem number 10
	fbSubsystem10: FB_ProBoxSubsystem;
	END_VAR VAR_GLOBAL CONSTANT NUMBERS_OF_ETHERCAT_SLAVE_DIAG: int :=50; //Number of EtherCAT Slaves;
END_VAR

// ---- 10_Project/10_App/12_FlowControl/00_GVLs/FlowControl.TcGVL
///Automatically created by BoxConfigurator
VAR_GLOBAL
	///Main merging service
	fbMergingService: FB_MergingService;
	///Main routing service
	fbRoutingService: FB_RoutingService;
END_VAR

// ---- 10_Project/11_Emu/10_Config/00_GVLs/GroupsEmulation.TcGVL
///Automatically generated by BoxConfigurator 
VAR_GLOBAL
	fbSG_001_Emulation                : FB_ProBOXSG_Emulation;
	fbSG_002_Emulation                : FB_ProBOXSG_Emulation;
END_VAR

// ---- 10_Project/11_Emu/10_Config/00_GVLs/PositionsEmulation.TcGVL
///Automatically generated by BoxConfigurator 
VAR_GLOBAL
	fbEL_10_001_0200_00_0_Emulation         : FB_ProBoxElementMotorEmulation;
	fbF_10_001_0200_01_0_Emulation          : FB_ProBoxStraightTransportEmulation;
	fbF_10_001_0200_02_0_Emulation          : FB_InOutFeedAddonEmulation;
	fbEL_10_001_0201_00_0_Emulation         : FB_ProBoxElementMotorEmulation;
	fbF_10_001_0201_01_0_Emulation          : FB_LowLiftUnitEmulation;
	fbEL_10_001_0202_00_0_Emulation         : FB_ProBoxElementMotorEmulation;
	fbF_10_001_0202_01_0_Emulation          : FB_ProBoxStraightTransportEmulation;
	fbEL_10_001_0203_00_0_Emulation         : FB_ProBoxElementMotorEmulation;
	fbF_10_001_0203_01_0_Emulation          : FB_ProBoxStraightTransportEmulation;
	fbF_10_001_0203_02_0_Emulation          : FB_ProfileCheckAddonEmulation;
	fbF_10_001_0203_03_0_Emulation          : FB_SickScannerAddonEmulation;
	fbF_10_001_0203_04_0_Emulation          : FB_TLB4WeightAddonEmulation;
	fbF_10_001_0203_05_0_Emulation          : FB_PalletCheckAddonEmulation;
	fbEL_10_001_0204_00_0_Emulation         : FB_ProBoxElementMotorEmulation;
	fbF_10_001_0204_01_0_Emulation          : FB_TurnTableEmulation;
	fbEL_10_001_0205_00_0_Emulation         : FB_ProBoxElementMotorEmulation;
	fbEL_10_001_0207_00_0_Emulation         : FB_ProBoxElementMotorEmulation;
	fbF_10_001_0207_01_0_Emulation          : FB_ProBoxStraightTransportEmulation;
	fbF_10_001_0207_02_0_Emulation          : FB_PalletMagazineAddonEmulation;
	fbEL_10_001_0208_00_0_Emulation         : FB_ProBoxElementMotorEmulation;
	fbF_10_001_0208_01_0_Emulation          : FB_ProBoxStraightTransportEmulation;
	fbEL_10_001_0209_00_0_Emulation         : FB_ProBoxElementMotorEmulation;
	fbF_10_001_0209_01_0_Emulation          : FB_TransferUnitEmulation;
	fbEL_10_001_0211_00_0_Emulation         : FB_ProBoxElementMotorEmulation;
	fbF_10_001_0211_01_0_Emulation          : FB_ProBoxStraightTransportEmulation;
	fbEL_10_001_0212_00_0_Emulation         : FB_ProBoxElementMotorEmulation;
	fbF_10_001_0212_01_0_Emulation          : FB_TransferUnitEmulation;
	fbEL_10_001_0213_00_0_Emulation         : FB_ProBoxElementMotorEmulation;
	fbF_10_001_0213_01_0_Emulation          : FB_ProBoxStraightTransportEmulation;
	fbF_10_001_0213_02_0_Emulation          : FB_PalletMagazineAddonEmulation;
	fbEL_10_001_0214_00_0_Emulation         : FB_ProBoxElementMotorEmulation;
	fbF_10_001_0214_01_0_Emulation          : FB_ProBoxStraightTransportEmulation;
	fbEL_10_001_0215_00_0_Emulation         : FB_ProBoxElementMotorEmulation;
	fbF_10_001_0215_01_0_Emulation          : FB_ProBoxStraightTransportEmulation;
	fbF_10_001_0215_02_0_Emulation          : FB_ProBoxStraightTransportEmulation;
	fbF_10_001_0215_03_0_Emulation          : FB_CraneXoverAddonEmulation;
	fbEL_10_001_0216_00_0_Emulation         : FB_ProBoxElementMotorEmulation;
	fbF_10_001_0216_01_0_Emulation          : FB_ProBoxStraightTransportEmulation;
	fbF_10_001_0216_02_0_Emulation          : FB_CraneXoverAddonEmulation;
	fbEL_10_001_0217_00_0_Emulation         : FB_ProBoxElementMotorEmulation;
	fbF_10_001_0217_01_0_Emulation          : FB_ProBoxStraightTransportEmulation;
	fbEL_10_001_0218_00_0_Emulation         : FB_ProBoxElementMotorEmulation;
	fbF_10_001_0218_01_0_Emulation          : FB_ProBoxStraightTransportEmulation;
	fbEL_10_001_0219_00_0_Emulation         : FB_ProBoxElementMotorEmulation;
	fbF_10_001_0219_01_0_Emulation          : FB_ProBoxStraightTransportEmulation;
	fbEL_10_001_0220_00_0_Emulation         : FB_ProBoxElementMotorEmulation;
	fbF_10_001_0220_01_0_Emulation          : FB_ProBoxStraightTransportEmulation;
	fbEL_10_001_0221_00_0_Emulation         : FB_ProBoxElementMotorEmulation;
	fbF_10_001_0221_01_0_Emulation          : FB_TransferUnitEmulation;
	fbEL_10_001_0222_00_0_Emulation         : FB_ProBoxElementMotorEmulation;
	fbF_10_001_0222_01_0_Emulation          : FB_TransferUnitEmulation;
	fbEL_10_001_0223_00_0_Emulation         : FB_ProBoxElementMotorEmulation;
	fbEL_10_001_0225_00_0_Emulation         : FB_ProBoxElementMotorEmulation;
	fbF_10_001_0225_01_0_Emulation          : FB_ProBoxStraightTransportEmulation;
	fbEL_10_001_0226_00_0_Emulation         : FB_ProBoxElementMotorEmulation;
	fbF_10_001_0226_01_0_Emulation          : FB_ProBoxStraightTransportEmulation;
	fbEL_10_001_0227_00_0_Emulation         : FB_ProBoxElementMotorEmulation;
	fbF_10_001_0227_01_0_Emulation          : FB_ProBoxStraightTransportEmulation;
	fbEL_10_001_0230_00_0_Emulation         : FB_ProBoxElementMotorEmulation;
	fbF_10_001_0230_01_0_Emulation          : FB_TransferCC_Emulation;
	fbEL_10_001_0232_00_0_Emulation         : FB_ProBoxElementMotorEmulation;
	fbF_10_001_0232_01_0_Emulation          : FB_ProBoxStraightTransportEmulation;
	fbF_10_001_0232_02_0_Emulation          : FB_InOutFeedAddonEmulation;
	fbEL_10_001_0233_00_0_Emulation         : FB_ProBoxElementMotorEmulation;
	fbF_10_001_0233_01_0_Emulation          : FB_ProBoxStraightTransportEmulation;
	fbEL_10_002_0206_00_0_Emulation         : FB_ProBoxElementMotorEmulation;
	fbF_10_002_0206_01_0_Emulation          : FB_ProBoxStraightTransportEmulation;
END_VAR

// ---- 10_Project/11_Emu/10_Config/00_GVLs/SubsystemEmulation.TcGVL
///Automatically created by BoxConfigurator
VAR_GLOBAL
	///Subsystem number 10 emulation
	fbSubsystem10_Emulation: FB_ProBoxSubsystemEmulation;
END_VAR

// ---- 20_Product/10_BCF/10_Base/00_GVLs/GVR_Table.TcGVL
(**************************************************************************************
 * 	Application		:	BoxControl Framework
 *	Revision		:	$Revision: 404529 $
 *	Revision date	:	$Date: 2018-04-23 08:21:38 +0200 (Mo., 23 Apr 2018) $
 *	Last changed by	:	$Author: b7bolm $
 *	URL				:	$URL: http://almscdc.swisslog.com/repo/SWPD/Development/BoxControlFramework/20_Release/trunk/01_Software/BCF/BCF/JumpStart/20_Product/10_App/10_Base/10_Lib/00_GVLs/GVR_Table.TcGVL $
 *
 *	Purpose			:	GVR signals - Separated due to debug reasons.
 *
 * ------------------------------------------------------------------------------------
 *	Copyright Swisslog [IP AG], Switzerland. All rights reserved.
 * 
 * ------------------------------------------------------------------------------------
 *	
 * 	Revision History: 
 *
 * 	VERSION			DATE			INITIALS			DESCRIPTION
 *	0.1				01.01.2001		swl					Example
 *
 **************************************************************************************)

VAR_GLOBAL CONSTANT
	NUMBER_OF_GVR_SIGNALS			: INT := 9999; // Number of ISR signals, max 9999 
END_VAR
 
VAR_GLOBAL
	GlobalVariable					: ARRAY[0..NUMBER_OF_GVR_SIGNALS, 0..9] OF DINT; // Array for GVR telegram
END_VAR

// ---- 20_Product/10_BCF/10_Base/00_GVLs/ISR_Table.TcGVL
(**************************************************************************************
 * 	Application		:	BoxControl Framework
 *	Revision		:	$Revision: 404529 $
 *	Revision date	:	$Date: 2018-04-23 08:21:38 +0200 (Mo., 23 Apr 2018) $
 *	Last changed by	:	$Author: b7bolm $
 *	URL				:	$URL: http://almscdc.swisslog.com/repo/SWPD/Development/BoxControlFramework/20_Release/trunk/01_Software/BCF/BCF/JumpStart/20_Product/10_App/10_Base/10_Lib/00_GVLs/ISR_Table.TcGVL $
 *
 *	Purpose			:	ISR signals - Separated due to debug reasons.
 *
 * ------------------------------------------------------------------------------------
 *	Copyright Swisslog [IP AG], Switzerland. All rights reserved.
 * 
 * ------------------------------------------------------------------------------------
 *	
 * 	Revision History: 
 *
 * 	VERSION			DATE			INITIALS			DESCRIPTION
 *	0.1				01.01.2001		swl					Example
 *
 **************************************************************************************)

VAR_GLOBAL CONSTANT
	NUMBER_OF_ISR_SIGNALS			: INT := 9999; // Number of ISR signals, max 9999 
	NUMBER_OF_ISR_DATA_LENGTH		: INT := 99; // Max length of data
END_VAR
 
VAR_GLOBAL
	ISR_SignalType					: ARRAY [0..2] OF ST_ISR_Table;	
END_VAR

// ---- 20_Product/10_BCF/10_Base/00_GVLs/RegistryEmulation.TcGVL
(**************************************************************************************
 * 	Application		:	BoxControl Framework
 *	Revision		:	$Revision: 404529 $
 *	Revision date	:	$Date: 2018-04-23 08:21:38 +0200 (Mo., 23 Apr 2018) $
 *	Last changed by	:	$Author: b7bolm $
 *	URL				:	$URL: http://almscdc.swisslog.com/repo/SWPD/Development/BoxControlFramework/20_Release/trunk/01_Software/BCF/BCF/JumpStart/20_Product/11_Emu/10_Base/10_Lib/00_GVLs/RegistryEmulation.TcGVL $
 *
 *	Purpose			:	Global registration. All types use the same. (Emulation)
 *
 * ------------------------------------------------------------------------------------
 *	Copyright Swisslog [IP AG], Switzerland. All rights reserved.
 * 
 * ------------------------------------------------------------------------------------
 *	
 * 	Revision History: 
 *
 * 	VERSION			DATE			INITIALS			DESCRIPTION
 *	0.1				01.01.2001		swl					Example
 *
 **************************************************************************************)
VAR_GLOBAL
	FunctionRegistryEmulation	: ARRAY[E_FunctionNumber.F_BEGIN_FUNCTION..E_FunctionNumber.F_END_EXTERN_FUNCTION -1] OF ST_FunctionRegistryConvEmulation; // Function registry
	ElementRegistryEmulation 	: ARRAY[E_ElementNumber.E_BEGIN_ELEMENT..E_ElementNumber.E_END_ELEMENT -1] OF ST_ElementRegistryConvEmulation; // Element registry 
	GroupRegistryEmulation 		: ARRAY[E_GroupNumber.G_BEGIN_GROUP..E_GroupNumber.G_END_GROUP -1] OF ST_GroupRegistryConvEmulation; // Group registry 
	SubsystemRegistryEmulation	: ST_SubsystemRegistryConvEmulation; // Subsystem registry	
END_VAR

// ---- 20_Product/10_BCF/10_Base/00_GVLs/SDI_Table.TcGVL
(**************************************************************************************
 * 	Application		:	BoxControl Framework
 *	Revision		:	$Revision: 404529 $
 *	Revision date	:	$Date: 2018-04-23 08:21:38 +0200 (Mo., 23 Apr 2018) $
 *	Last changed by	:	$Author: b7bolm $
 *	URL				:	$URL: http://almscdc.swisslog.com/repo/SWPD/Development/BoxControlFramework/20_Release/trunk/01_Software/BCF/BCF/JumpStart/20_Product/10_App/10_Base/10_Lib/00_GVLs/SDI_Table.TcGVL $
 *
 *	Purpose			:	SDO signals - separated due to debug reasons.
 *
 * ------------------------------------------------------------------------------------
 *	Copyright Swisslog [IP AG], Switzerland. All rights reserved.
 * 
 * ------------------------------------------------------------------------------------
 *	
 * 	Revision History: 
 *
 * 	VERSION			DATE			INITIALS			DESCRIPTION
 *	0.1				01.01.2001		swl					Example
 *
 **************************************************************************************)
VAR_GLOBAL CONSTANT
	NUMBER_OF_SDI_SIGNALS			: INT := 9999; // Number of SDI signals, max 9999 
END_VAR

VAR_GLOBAL
	SDISignalNumber					: ARRAY [0..NUMBER_OF_SDI_SIGNALS] OF ST_SDI_TABLE; // SDI table
END_VAR

// ---- 20_Product/10_BCF/10_Base/00_GVLs/SDO_Table.TcGVL
(**************************************************************************************
 * 	Application		:	BoxControl Framework
 *	Revision		:	$Revision: 404529 $
 *	Revision date	:	$Date: 2018-04-23 08:21:38 +0200 (Mo., 23 Apr 2018) $
 *	Last changed by	:	$Author: b7bolm $
 *	URL				:	$URL: http://almscdc.swisslog.com/repo/SWPD/Development/BoxControlFramework/20_Release/trunk/01_Software/BCF/BCF/JumpStart/20_Product/10_App/10_Base/10_Lib/00_GVLs/SDO_Table.TcGVL $
 *
 *	Purpose			:	SDO signals - Separated due to debug reasons.
 *
 * ------------------------------------------------------------------------------------
 *	Copyright Swisslog [IP AG], Switzerland. All rights reserved.
 * 
 * ------------------------------------------------------------------------------------
 *	
 * 	Revision History: 
 *
 * 	VERSION			DATE			INITIALS			DESCRIPTION
 *	0.1				01.01.2001		swl					Example
 *
 **************************************************************************************)

VAR_GLOBAL CONSTANT
	NUMBER_OF_SDO_SIGNALS			: INT := 9999; // Number of SDO signals, max 9999 
END_VAR
 
VAR_GLOBAL
	SDOSignalNumber					: ARRAY [0..NUMBER_OF_SDO_SIGNALS] OF BOOL; // SDO table
END_VAR

// ---- 20_Product/10_BCF/10_Base/00_GVLs/System.TcGVL
(**************************************************************************************
 * 	Application		:	BoxControl Framework
 *	Revision		:	$Revision: 404529 $
 *	Revision date	:	$Date: 2018-04-23 08:21:38 +0200 (Mo., 23 Apr 2018) $
 *	Last changed by	:	$Author: b7bolm $
 *	URL				:	$URL: http://almscdc.swisslog.com/repo/SWPD/Development/BoxControlFramework/20_Release/trunk/01_Software/BCF/BCF/JumpStart/20_Product/10_App/10_Base/10_Lib/00_GVLs/System.TcGVL $
 *
 *	Purpose			:	Base global variables.
 *
 * ------------------------------------------------------------------------------------
 *	Copyright Swisslog [IP AG], Switzerland. All rights reserved.
 * 
 * ------------------------------------------------------------------------------------
 *	
 * 	Revision History: 
 *
 * VERSION DATE         INITIALS     DESCRIPTION
 * 0.0     DD.MM.YYYY   (name)       (explain customized modifications)
 *
 **************************************************************************************)
VAR_GLOBAL CONSTANT
	NAME_LENGTH						: INT := 20; // String length Subsystem, group, element and zone name  
	DEBUGSOURCELENGTH 				: INT := 255; // String length debug source 
	DEBUGMESSAGELENGTH 				: INT := 250; // String length debug message 
	ERROR_PARAM_STRINGLENGTH		: INT := 50; // Error param string length	
	NUMBER_OF_KEYVALUE_PAIRS_VIR	: INT := 99; // Maximum number of KeyValue-Pairs in a visualization report
	KEY_LENGTH						: INT := 30; // Maximum  key length for visualization report
	VALUE_LENGTH					: INT := 18; // Maximum value length for visualization report
	NUMBER_OF_KEYS_VIQ				: INT := 99; // Maximum number of Keys in a visualization request
	CM_MAX_NUMBER_Of_ENTRIES		: INT := 99; //  Number of Entries in one report. 
	CM_VARIABLENAME_STRINGLENGTH	: INT := 20; // DA Variable Name Length 20 char
	CM_VARIABLE_STRINGLENGTH		: INT := 20; // DA Variable Length 20 char
	CM_TIMESTAMP_MS_STRINGLENGTH	: INT := 23; // DA Timestamp with MS Length 23 char
	CM_DATASET_STRINGLENGTH			: INT := 47; // DA Length of one Data set 23 char
END_VAR

VAR_GLOBAL
	fbSystemTime					: NT_GetTime; // Get System time 
	TimeStampDT						: DATE_AND_TIME; // Current Time Stamp DT 
	ActCycleTime					: DINT; // Calculated cycle time in micro seconds
	fbBlink_100ms					: FB_GeneratePulse := (Start := TRUE, PulseTimeOn := T#100MS, PulseTimeOff := T#100MS); // Blink 100ms
	fbBlink_500ms					: FB_GeneratePulse := (Start := TRUE, PulseTimeOn := T#500MS, PulseTimeOff := T#500MS); // Blink 500ms
	fbBlink_1s						: FB_GeneratePulse := (Start := TRUE, PulseTimeOn := T#1S, PulseTimeOff := T#1S); // Blink 1s
	fbSocketCloseAll				: FB_SocketCloseAll := (sSrvNetID := '', tTimeout := DEFAULT_ADS_TIMEOUT); // Closing all sockets
	fbMFCS_Channel					: ARRAY [E_MFCS_Channel.BEGIN_CHANNEL .. E_MFCS_Channel.END_CHANNEL] OF ITF_MFCS; // MFCS connections
	fbITC_Manager					: ITF_ITC;
	fbDebugMsgManager				: FB_DebugMsgManager; // Debug message manager
	fbFormatString					: FB_FormatString; // Building strings with arguments
	TimeStampString					: STRING(23); // Current Time Stamp as String 
END_VAR

// ---- 20_Product/10_BCF/10_Base/00_GVLs/SystemEmulation.TcGVL
(**************************************************************************************
 * 	Application		:	BoxControl Framework
 *	Revision		:	$Revision: 404529 $
 *	Revision date	:	$Date: 2018-04-23 08:21:38 +0200 (Mo., 23 Apr 2018) $
 *	Last changed by	:	$Author: b7bolm $
 *	URL				:	$URL: http://almscdc.swisslog.com/repo/SWPD/Development/BoxControlFramework/20_Release/trunk/01_Software/BCF/BCF/JumpStart/20_Product/11_Emu/10_Base/10_Lib/00_GVLs/SystemEmulation.TcGVL $
 *
 *	Purpose			:	Base emulation global variables.
 *
 * ------------------------------------------------------------------------------------
 *	Copyright Swisslog [IP AG], Switzerland. All rights reserved.
 * 
 * ------------------------------------------------------------------------------------
 *	
 * 	Revision History: 
 *
 * 	VERSION			DATE			INITIALS			DESCRIPTION
 *	0.1				01.01.2001		swl					Example
 *
 **************************************************************************************)
VAR_GLOBAL
	fbMFCS_ChannelEmulation		: ARRAY [E_MFCS_Channel.BEGIN_CHANNEL .. E_MFCS_Channel.END_CHANNEL] OF ITF_MFCS_Emulation; // MFCS connections
	fbITC_ManagerEmulation		: ITF_ITC_Emulation;
END_VAR

// ---- 20_Product/10_BCF/10_Base/11_Com/12_DebugMsg/00_GVLs/DebugTextBlocks.TcGVL
(**************************************************************************************
 * 	Application		:	BoxControl Framework
 *	Revision		:	$Revision: 475016 $
 *	Revision date	:	$Date: 2021-04-09 08:29:02 +0200 (fre, 09 apr 2021) $
 *	Last changed by	:	$Author: d7mangc $
 *	URL				:	$URL: http://almscdc.swisslog.com/repo/SWPD/Development/BoxControlFramework/20_Release/tags/R1.12.0/01_Software/BCF/BCF/JumpStart/20_Product/10_BCF/10_Base/11_Com/12_DebugMsg/00_GVLs/DebugTextBlocks.TcGVL $
 *
 *	Purpose			:	Common text blocks for debug messages
 *                      to ensure that uniform text is used in all messages and can be searched for and filtered more easily
 *
 * ------------------------------------------------------------------------------------
 *	Copyright Swisslog [IP AG], Switzerland. All rights reserved.
 * 
 * ------------------------------------------------------------------------------------
 *	
 * 	Revision History: 
 *
 * VERSION DATE         INITIALS     DESCRIPTION
 * 0.0     DD.MM.YYYY   (name)       (explain customized modifications)
 *
 **************************************************************************************)

{attribute 'strict'}
{attribute 'qualified_only'}                 //          1         2         3
VAR_GLOBAL CONSTANT                          // 123456789012345678901234567890
	ASSIGNMENTID		: STRING[19]		:= ',  AssignmentID = ';
	CURRENT				: STRING[15]		:= ',  current = ';
	DESTINATION			: STRING[19]		:= ',  destination = ';
	DRIVE				: STRING[15]		:= ',  drive = ';
	ENDLENGTH			: STRING[19]		:= ',  end length = ';
	EXPECTED			: STRING[15]		:= ',  expected = ';
	FREE				: STRING[11]		:= ',  free = ';
	FOLDER				: STRING[15]		:= ',  folder = ';
	FUNCTIONNBR			: STRING[15]		:= ',  function = ';
	LABEL				: STRING[11]		:= ',  label = ';
	LENGTH				: STRING[15]		:= ',  length = ' ;
	MISSED				: STRING[15]		:= ',  missed = ';
	OCCUPIED			: STRING[15]		:= ',  occupied = ';
	ORIGIN				: STRING[15]		:= ',  origin = ';
	POSITION			: STRING[15]		:= ',  position = ';
	RANGE				: STRING[15]		:= ',  range = 0..';
	SPEED				: STRING[11]		:= ',  speed = ';
	STOPDELAY 			: STRING[19]		:= ',  stopp delay = ';
	TELEGRAM			: STRING[15]		:= ',  telegram = ';
	TIMEOUT				: STRING[15]		:= ',  timeout = ';
	TOTAL				: STRING[15]		:= ',  total = ';
	TU_DATA_INDEX		: STRING[19]		:= ',  TU_DataIndex = ';
	TUID				: STRING[15]		:= ',  TuID = ';
	USAGE				: STRING[11]		:= ',  usage = ';
	USED				: STRING[11]		:= ',  used = ';
	ZONENBR				: STRING[11]		:= ',  zone = ';
END_VAR

// ---- 20_Product/10_BCF/11_Conv/10_Base/00_GVLs/Conveyor.TcGVL
(**************************************************************************************
 * 	Application		:	BoxControl Framework
 *	Revision		:	$Revision: 412414 $
 *	Revision date	:	$Date: 2018-08-17 07:57:24 +0200 (Fr., 17 Aug 2018) $
 *	Last changed by	:	$Author: d7herza $
 *	URL				:	$URL: http://almscdc.swisslog.com/repo/SWPD/Development/BoxControlFramework/20_Release/trunk/01_Software/BCF/BCF/JumpStart/20_Product/10_App/10_Base/10_Lib/10_Conv/00_GVLs/Conveyor.TcGVL $
 *
 *	Purpose			:	Global variables : Conveyor
 *
 * ------------------------------------------------------------------------------------
 *	Copyright Swisslog [IP AG], Switzerland. All rights reserved.
 * 
 * ------------------------------------------------------------------------------------
 *	
 * 	Revision History: 
 *
 * 	VERSION			DATE			INITIALS			DESCRIPTION
 *	0.1				01.01.2001		swl					Example
 *
 **************************************************************************************)
VAR_GLOBAL
	fbGroupManager						: FB_GroupManager; // Group manager
	//fbITC_ManagerConveyor 				: FB_ITC_Conveyor;	Overloaded by ProBox fb_PB_ITC_ManagerConveyor
	fbMFCS_SIS_AM						: FB_SIS_MsgManager_6_1; // SIS AM
	fbMFCS_SIS_SPOC						: FB_SIS_MsgManager_6_1; // SIS SPOC
	fbMFCS_LOG							: FB_SIS_MsgManager_6_1; // SIS LOG
	fbMFCS_SIS_CM						: FB_SIS_MsgManager_6_1; // SIS CM
	fbSTI_Channels						: ARRAY[E_FunctionNumber.F_BEGIN_EXTERN_FUNCTION .. E_FunctionNumber.F_END_EXTERN_FUNCTION] OF ST_STI_Channel;
	ExternalDestinationTable			: ARRAY[E_FunctionNumber.F_BEGIN_VIRTUAL_FUNCTION ..E_FunctionNumber.F_END_VIRTUAL_FUNCTION , 1..Conveyor.NUMBER_OF_EXT_DESTINATIONS] OF ST_ExternalDestination;
END_VAR

VAR_GLOBAL CONSTANT
	TU_ID_UNKNOWN						: STRING(TU_ID_STRINGLENGTH) := '999999999999999999'; // String for unkwnon TU-ID  
	ASSIGNMENT_ID_UNKNOWN				: UDINT := 99999999; // String for unkwnon Assignment-ID  
	NUMBER_OF_TU_DATA					: DINT := 5000; // Size of the TU-Data 
	NUMBER_OF_ADDON_FUNCTIONS			: INT := 5; // Number of Addons per function
	NUMBER_OF_ZONES_PER_FUNCTION		: INT := 4; // Max number of zones per element function
	NUMBER_OF_FUNCTIONS_PER_ELEMENT		: INT := 8; // Possible element functions on a certain element
	NUMBER_OF_ACTIONS					: INT := 10; // Number of input or output actions of a windows tracking. 	
	NUMBER_OF_WINDOWS					: WORD := 1024; // Number of windows over the complete tracking length
	NUMBER_OF_TRACKING_ZONES			: INT := 1024; // Number of zones over the complete tracking length
	NUMBER_OF_EXT_DESTINATIONS			: INT := 10; // Number of external destinations per virtual destination
	TU_ID_STRINGLENGTH					: INT := 18; // Number of characters for the TU-ID 
	LABEL_LENGTH						: INT := 20; // Label length
	NUMBER_OF_STI						: INT := 4; // Number of Subsystem transport interfaces
	POSITION_STRINGLENGTH				: INT := 12; // PositionName MM-000-0000-000
	ORIENTATION_STRINGLENGTH			: INT := 3; // String length	
	TU_DATA_LIFETIME					: TIME := T#3D; // Delets the the TU-Data after this time 
	NUMBER_OF_DESTINATIONS				: INT := 2; // Number of destinations in the TU-Data 
	ASSIGNMENT_ID_STRINGLENGTH			: INT := 8; // Assignment ID string
	NUMBER_OF_ERROR_SETS				: INT := 8; // Number of possible error sets per position
	//NUMBERS_OF_ETHERCAT_SLAVE_DIAG		: INT := 50; // Number of EtherCAT Slaves
    MAX_LOADING                  	  	: INT := 50; // maximum weight of a transport unit [kg] 
	NUMBER_OF_COMMAND_ARGS				: INT := 99; // Maximum number of custom param counts 
	ROBOT_COMMAND_LENGTH				: INT := 20000; // Lengt of a robot command
	GATHERED_DATA_VALUE					: INT := 20;// 20 Character String;
	KEY_STRINGLENGTH					: INT := 30; // key length
END_VAR

// ---- 20_Product/10_BCF/11_Conv/10_Base/00_GVLs/ExecutionTimeTable.TcGVL
{attribute 'qualified_only'}
(**************************************************************************************
 * 	Application		:	BoxControl Framework
 *	Revision		:	$Revision: 404529 $
 *	Revision date	:	$Date: 2018-04-23 08:21:38 +0200 (Mo., 23 Apr 2018) $
 *	Last changed by	:	$Author: b7bolm $
 *	URL				:	$URL: http://almscdc.swisslog.com/repo/SWPD/Development/BoxControlFramework/20_Release/trunk/01_Software/BCF/BCF/JumpStart/20_Product/10_App/10_Base/10_Lib/10_Conv/00_GVLs/ExecutionTimeTable.TcGVL $
 *
 *	Purpose			:	Execution time of all position calls
 *
 * ------------------------------------------------------------------------------------
 *	Copyright Swisslog [IP AG], Switzerland. All rights reserved.
 * 
 * ------------------------------------------------------------------------------------
 *	
 * 	Revision History: 
 *
 * 	VERSION			DATE			INITIALS			DESCRIPTION
 *	0.1				01.01.2001		swl					Example
 *
 **************************************************************************************)
VAR_GLOBAL
	MFCS_Channels		: ARRAY [E_MFCS_Channel.BEGIN_CHANNEL .. E_MFCS_Channel.END_CHANNEL] OF ST_ExecutionTime;
	DebugMsgManager		: ST_ExecutionTime;
	ITC_Manager			: ST_ExecutionTime;
	Subsystem			: ST_ExecutionTime;
	Groups				: ARRAY [E_GroupNumber.G_BEGIN_GROUP .. E_GroupNumber.G_END_GROUP] OF ST_ExecutionTime;
	Elements			: ARRAY [E_ElementNumber.E_BEGIN_ELEMENT .. E_ElementNumber.E_END_ELEMENT] OF ST_ExecutionTime;
	Functions			: ARRAY [E_FunctionNumber.F_BEGIN_FUNCTION .. E_FunctionNumber.F_END_FUNCTION] OF ST_ExecutionTime;
END_VAR

// ---- 20_Product/10_BCF/11_Conv/10_Base/00_GVLs/Registry.TcGVL
(**************************************************************************************
 * 	Application		:	BoxControl Framework
 *	Revision		:	$Revision: 404529 $
 *	Revision date	:	$Date: 2018-04-23 08:21:38 +0200 (Mo., 23 Apr 2018) $
 *	Last changed by	:	$Author: b7bolm $
 *	URL				:	$URL: http://almscdc.swisslog.com/repo/SWPD/Development/BoxControlFramework/20_Release/trunk/01_Software/BCF/BCF/JumpStart/20_Product/10_App/10_Base/10_Lib/10_Conv/00_GVLs/Registry.TcGVL $
 *
 *	Purpose			:	Global registration. All types use the same
 *
 * ------------------------------------------------------------------------------------
 *	Copyright Swisslog [IP AG], Switzerland. All rights reserved.
 * 
 * ------------------------------------------------------------------------------------
 *	
 * 	Revision History: 
 *
 * 	VERSION			DATE			INITIALS			DESCRIPTION
 *	0.1				01.01.2001		swl					Example
 *
 **************************************************************************************)
VAR_GLOBAL
	FunctionRegistry	: ARRAY[E_FunctionNumber.F_BEGIN_FUNCTION..E_FunctionNumber.F_END_EXTERN_FUNCTION -1] OF ST_FunctionRegistryConv; // Function registry
	ElementRegistry 	: ARRAY[E_ElementNumber.E_BEGIN_ELEMENT..E_ElementNumber.E_END_ELEMENT -1] OF ST_ElementRegistryConv; // Element registry 
	GroupRegistry 		: ARRAY[E_GroupNumber.G_BEGIN_GROUP..E_GroupNumber.G_END_GROUP -1] OF ST_GroupRegistryConv; // Group registry 
	SubsystemRegistry	: ST_SubsystemRegistryConv; // Subsystem registry	
END_VAR

// ---- 20_Product/10_BCF/11_Conv/10_Base/00_GVLs/TU_Table.TcGVL
(**************************************************************************************
 * 	Application		:	BoxControl Framework
 *	Revision		:	$Revision: 404529 $
 *	Revision date	:	$Date: 2018-04-23 08:21:38 +0200 (Mo., 23 Apr 2018) $
 *	Last changed by	:	$Author: b7bolm $
 *	URL				:	$URL: http://almscdc.swisslog.com/repo/SWPD/Development/BoxControlFramework/20_Release/trunk/01_Software/BCF/BCF/JumpStart/20_Product/10_App/10_Base/10_Lib/10_Conv/00_GVLs/TU_Table.TcGVL $
 *
 *	Purpose			:	Global variables : Conveyor TU Data
 *
 * ------------------------------------------------------------------------------------
 *	Copyright Swisslog [IP AG], Switzerland. All rights reserved.
 * 
 * ------------------------------------------------------------------------------------
 *	
 * 	Revision History: 
 *
 * 	VERSION			DATE			INITIALS			DESCRIPTION
 *	0.1				01.01.2001		swl					Example
 *
 **************************************************************************************)
VAR_GLOBAL PERSISTENT
	TU_DataTable 	: ARRAY[0..Conveyor.NUMBER_OF_TU_DATA] OF ST_TU_Data; // Contains all TU-data
END_VAR

// ---- 20_Product/10_BCF/11_Conv/10_Base/ConveyorEmulation.TcGVL
(**************************************************************************************
 * 	Application		:	BoxControl Framework
 *	Revision		:	$Revision: 404529 $
 *	Revision date	:	$Date: 2018-04-23 08:21:38 +0200 (Mo., 23 Apr 2018) $
 *	Last changed by	:	$Author: b7bolm $
 *	URL				:	$URL: http://almscdc.swisslog.com/repo/SWPD/Development/BoxControlFramework/20_Release/trunk/01_Software/BCF/BCF/JumpStart/20_Product/11_Emu/10_Base/10_Lib/10_Conv/00_GVLs/ConveyorEmulation.TcGVL $
 *
 *	Purpose			:	Conveyor emulation global variables.
 *
 * ------------------------------------------------------------------------------------
 *	Copyright Swisslog [IP AG], Switzerland. All rights reserved.
 * 
 * ------------------------------------------------------------------------------------
 *	
 * 	Revision History: 
 *
 * 	VERSION			DATE			INITIALS			DESCRIPTION
 *	0.1				01.01.2001		swl					Example
 *
 **************************************************************************************)
VAR_GLOBAL
	EmulationActive					: BOOL;  // Emulation is active
	fbMFCS_SIS_AM_Emulation			: FB_SIS_MsgManager_6_1_Emulation; // SIS AM Emulation
	fbMFCS_SIS_SPOC_Emulation		: FB_SIS_MsgManager_6_1_Emulation; // SIS SPOC Emulation
	fbMFCS_SIS_LOG_Emulation		: FB_SIS_MsgManager_6_1_Emulation; // SIS LOG Emulation
	fbITC_ConveyorEmulation 		: FB_ITC_ConveyorEmulation;
	fbSTI_ChannelsEmulation			: ARRAY [E_FunctionNumber.F_BEGIN_EXTERN_FUNCTION .. E_FunctionNumber.F_END_EXTERN_FUNCTION] OF ST_STI_ChannelEmulation;
END_VAR

VAR_GLOBAL CONSTANT
	LABEL_STRING_LENGTH				: INT := 80; // 80 digit label
	NUMBER_OF_TU_PER_FUNCTION		: INT := 10; // Max number of TU's per element function
END_VAR

VAR_GLOBAL PERSISTENT
	TU_DataTableEmulation 			: ARRAY[0..Conveyor.NUMBER_OF_TU_DATA] OF ST_TU_DataEmulation; // Contains all TU-data
END_VAR

// ---- 20_Product/20_ProBox/10_Base/00_GVLs/PBTransportCtrl.TcGVL
{attribute 'qualified_only'}
VAR_GLOBAL	
	pbTransportControlDataEmpty 	: ST_TransportControlData; // Transport control data
	pbZoneSettingsEmpty				: ST_CFG_Zone;	
END_VAR

// ---- 20_Product/20_ProBox/10_Base/00_GVLs/ProBox_Conveyor.TcGVL
//{attribute 'qualified_only'}
VAR_GLOBAL
	fb_PB_ITC_ManagerConveyor 		: FB_PB_ITC_Conveyor;		
END_VAR

// ---- 20_Product/20_ProBox/30_Toolbox/70_Strategies/01_DUTs/GVL_Strategies.TcGVL
{attribute 'qualified_only'}
VAR_GLOBAL
	CONSTANT	 
	 MAX_TRANSFERUNITS		: INT := 30;	
END_VAR

// ---- 20_Product/30_Toolbox/16_Sequencing/00_GVLs/SequencingParameter.TcGVL
{attribute 'qualified_only'}
VAR_GLOBAL CONSTANT
	MAX_STREAMBUILDER_LIST		: INT := 200; // Max number of stored entries for a stream
	MAX_ESTIMATE_ALL_NEXT_LIST	: INT := 100; // Max entries for estimate next for all destination
	SCAN_ENTRIES_PER_CYCLE		: INT := 600; // Scanned TU entries per cycle
	DEFAULT_WARNING_TIME		: TIME := T#15M; // Default time to raise warning
	SEQ_VALIDATION_QUEUE		: UINT := 3; // Number of considered TU to be validated
	MAX_LIMITED_STREAM_LIST		: INT := 30; // Max number of stored entries for a limited stream	
	MAX_LANE_SIZE				: DINT := 10; // Max number of zones in a sequence conveyor lane			
END_VAR

// ---- 20_Product/30_Toolbox/17_WindowTracking/10_Core/00_GVLs/WindowTracking.TcGVL
{attribute 'qualified_only'}
VAR_GLOBAL CONSTANT
	MAX_NUMBER_OF_WINDOWS	: UINT := 2048; // Max number of tracking windows
	MAX_NUMBER_OF_ZONES		: UINT := MAX_NUMBER_OF_WINDOWS /2; // Max number of zones
END_VAR

// ---- 20_Product/10_BCF/10_Base/10_StateMachine/I_StateMachineTextCallback.TcIO
// callback event to retrieve state text
{attribute 'monitoring' := 'call'}
INTERFACE PUBLIC I_StateMachineTextCallback

// forwards state text to FB_StateMachine
METHOD PUBLIC M_GetStateText : A_StateText

VAR_INPUT
	StateMachine	: POINTER TO FB_StateMachine;	// requesting state machine instance
	StateNbr		: UINT;		                    // state number which text is requested
END_VAR
END_METHOD

END_INTERFACE

// ---- 20_Product/10_BCF/10_Base/11_Com/12_DebugMsg/20_TraceHandler/I_TraceHandler.TcIO
// writes traces into files, deletes too old files and monitors hdd usage
{attribute 'monitoring' := 'call'}
INTERFACE PUBLIC I_TraceHandler

// clears the internal fifo (all unwritten traces will be lost)
METHOD PUBLIC Clear

(********************************************************************************************************************************)
VAR_INPUT
END_VAR
END_METHOD

// HI = writing/deleting enabled
{attribute 'monitoring' := 'call'}
PROPERTY PUBLIC Enable : BOOL
GET
END_GET
SET
END_SET
END_PROPERTY

// folder to work within, folder must exist! (will only take effect when enabled is low)
{attribute 'monitoring' := 'call'}
PROPERTY PUBLIC Folder : A_TracePath
GET
END_GET
SET
END_SET
END_PROPERTY

// maximum file size in kilobytes
{attribute 'monitoring' := 'call'}
PROPERTY PUBLIC MaxFileSizeKB : WORD
GET
END_GET
SET
END_SET
END_PROPERTY

// HI = file is currently open
{attribute 'monitoring' := 'call'}
PROPERTY PUBLIC Opened : BOOL
GET
END_GET
END_PROPERTY

// puts a new trace line into the current file
METHOD PUBLIC Put

(********************************************************************************************************************************)
VAR_INPUT
  MsgType               : E_DebugMsgType                   := E_DebugMsgType.ERROR;
  Instance              : POINTER TO BYTE                  := 0;     // pointer to string
  Text                  : POINTER TO BYTE                  := 0;     // pointer to string
END_VAR
END_METHOD

// diagnosis & statisticals
{attribute 'monitoring' := 'call'}
PROPERTY PUBLIC Statistics : I_TraceHandlerStatistics
GET
END_GET
END_PROPERTY

END_INTERFACE

// ---- 20_Product/10_BCF/10_Base/11_Com/ITF_ITC.TcIO
INTERFACE ITF_ITC EXTENDS __System.IQueryInterface

METHOD M_AddData : BOOL
VAR_INPUT
	meChannelSrc	: E_MFCS_Channel;
	mMsgType		: INT;
	mpData			: PVOID;
	mLen			: UDINT;
END_VAR
END_METHOD

METHOD M_CallITC_Service : BOOL
VAR_INPUT
END_VAR
END_METHOD

METHOD M_Init : BOOL
(**************************************************************************************
 * 	Application		:	BoxControl Framework
 *	Revision		:	$Revision: 355272 $
 *	Revision date	:	$Date: 2015-09-23 11:26:06 +0200 (Wed, 23 Sep 2015) $
 *	Last changed by	:	$Author: b7bolm $
 *	URL				:	$URL: http://almscdc.swisslog.com/repo/SWPD/Development/BoxControlFramework/20_Release/trunk/01_Software/BoxControlFramework/BoxControlFramework/JumpStart/11_Library/10_Application/11_Communication/12_MFCS/11_SIS/11_SIS_6_0/FB_SIS_MsgManager_6_0.TcPOU $
 *
 *	Purpose			:	Initialize 
 *
 * ------------------------------------------------------------------------------------
 *	Copyright Swisslog [IP AG], Switzerland. All rights reserved.
 * 
 * ------------------------------------------------------------------------------------
 *	
 * 	Revision History: 
 *
 * 	VERSION			DATE			INITIALS			DESCRIPTION
 *	0.1				01.01.2001		swl					Example
 *
 **************************************************************************************)
VAR_INPUT
	mInit		: BOOL; // Force init
END_VAR
END_METHOD

METHOD M_SendData : BOOL
VAR_INPUT
	meChannel	: E_MFCS_Channel;
	mMsgType	: INT;
	mpData		: PVOID;
	mLen		: UDINT;
END_VAR
END_METHOD

END_INTERFACE

// ---- 20_Product/10_BCF/10_Base/11_Com/ITF_MFCS.TcIO
INTERFACE ITF_MFCS EXTENDS __System.IQueryInterface

METHOD M_BufferLevelAlarm : BOOL
VAR_INPUT
END_VAR
END_METHOD

METHOD M_BufferLevelWarning : BOOL
VAR_INPUT
END_VAR
END_METHOD

METHOD M_CallCommunicationService
(**************************************************************************************
 * 	Application		:	BoxControl Framework
 *	Revision		:	$Revision: 355272 $
 *	Revision date	:	$Date: 2015-09-23 11:26:06 +0200 (Wed, 23 Sep 2015) $
 *	Last changed by	:	$Author: b7bolm $
 *	URL				:	$URL: http://almscdc.swisslog.com/repo/SWPD/Development/BoxControlFramework/20_Release/trunk/01_Software/BoxControlFramework/BoxControlFramework/JumpStart/11_Library/10_Application/11_Communication/11_ITC/ITF_MsgManageable.TcIO $
 *
 *	Purpose			:	Interface for call communication service.
 *
 * ------------------------------------------------------------------------------------
 *	Copyright Swisslog [IP AG], Switzerland. All rights reserved.
 * 
 * ------------------------------------------------------------------------------------
 *	
 * 	Revision History: 
 *
 * 	VERSION			DATE			INITIALS			DESCRIPTION
 *	0.1				01.01.2001		swl					Example
 *
 **************************************************************************************)
VAR_INPUT
END_VAR
END_METHOD

METHOD M_GetReceivedData : ST_PointerSet
(**************************************************************************************
 * 	Application		:	BoxControl Framework
 *	Revision		:	$Revision: 355272 $
 *	Revision date	:	$Date: 2015-09-23 11:26:06 +0200 (Wed, 23 Sep 2015) $
 *	Last changed by	:	$Author: b7bolm $
 *	URL				:	$URL: http://almscdc.swisslog.com/repo/SWPD/Development/BoxControlFramework/20_Release/trunk/01_Software/BoxControlFramework/BoxControlFramework/JumpStart/11_Library/10_Application/11_Communication/11_ITC/ITF_MsgManageable.TcIO $
 *
 *	Purpose			:	Received data
 *
 * ------------------------------------------------------------------------------------
 *	Copyright Swisslog [IP AG], Switzerland. All rights reserved.
 * 
 * ------------------------------------------------------------------------------------
 *	
 * 	Revision History: 
 *
 * 	VERSION			DATE			INITIALS			DESCRIPTION
 *	0.1				01.01.2001		swl					Example
 *
 **************************************************************************************)
END_METHOD

METHOD M_Init : BOOL
(**************************************************************************************
 * 	Application		:	BoxControl Framework
 *	Revision		:	$Revision: 355272 $
 *	Revision date	:	$Date: 2015-09-23 11:26:06 +0200 (Wed, 23 Sep 2015) $
 *	Last changed by	:	$Author: b7bolm $
 *	URL				:	$URL: http://almscdc.swisslog.com/repo/SWPD/Development/BoxControlFramework/20_Release/trunk/01_Software/BoxControlFramework/BoxControlFramework/JumpStart/11_Library/10_Application/11_Communication/12_MFCS/11_SIS/11_SIS_6_0/FB_SIS_MsgManager_6_0.TcPOU $
 *
 *	Purpose			:	Initialize 
 *
 * ------------------------------------------------------------------------------------
 *	Copyright Swisslog [IP AG], Switzerland. All rights reserved.
 * 
 * ------------------------------------------------------------------------------------
 *	
 * 	Revision History: 
 *
 * 	VERSION			DATE			INITIALS			DESCRIPTION
 *	0.1				01.01.2001		swl					Example
 *
 **************************************************************************************)
VAR_INPUT
	mInit		: BOOL; // Force init
END_VAR
END_METHOD

METHOD M_IsConnected : BOOL
VAR_INPUT
END_VAR
END_METHOD

METHOD M_SendData : BOOL
VAR_INPUT
	meChannelSrc	: E_MFCS_Channel; // Source communicaton channel	
	mMsgType		: INT;
	mpData			: PVOID;
	mLen			: UDINT;
END_VAR
END_METHOD

END_INTERFACE

// ---- 20_Product/10_BCF/10_Base/11_Com/ITF_MFCS_Emulation.TcIO
INTERFACE ITF_MFCS_Emulation EXTENDS __SYSTEM.IQueryInterface

METHOD M_ProcessData : BOOL
(**************************************************************************************
 * 	Application		:	BoxControl Framework
 *	Revision		:	$Revision: 352632 $
 *	Revision date	:	$Date: 2015-07-20 08:49:54 +0200 (Mon, 20 Jul 2015) $
 *	Last changed by	:	$Author: b7bolm $
 *	URL				:	$URL: http://almscdc.swisslog.com/repo/SWPD/Development/BoxControlFramework/20_Release/trunk/01_Software/BoxControlFramework/BoxControlFramework/JumpStart/11_Library/10_Application/11_Communication/11_ITC/ITF_MsgManageable.TcIO $
 *
 *	Purpose			:	Process emulation data
 *
 * ------------------------------------------------------------------------------------
 *	Copyright Swisslog [IP AG], Switzerland. All rights reserved.
 * 
 * ------------------------------------------------------------------------------------
 *	
 * 	Revision History: 
 *
 * 	VERSION			DATE			INITIALS			DESCRIPTION
 *	0.1				01.01.2001		swl					Example
 *
 **************************************************************************************)
VAR_INPUT
	meChannelSrc	: E_MFCS_Channel; // MFCS Channel
	mData			: ST_PointerSet; // Data
END_VAR
END_METHOD

END_INTERFACE

// ---- 20_Product/10_BCF/11_Conv/11_Com/11_ITC/ITF_ITC_Emulation.TcIO
INTERFACE ITF_ITC_Emulation EXTENDS __System.IQueryInterface

METHOD M_AddData : BOOL
VAR_INPUT
	meChannelSrc	: E_MFCS_Channel;
	mMsgType		: INT;
	mpData			: PVOID;
	mLen			: UDINT;
END_VAR
END_METHOD

METHOD M_CallITC_Service : BOOL
VAR_INPUT
END_VAR
END_METHOD

END_INTERFACE

// ---- 20_Product/10_BCF/11_Conv/11_Com/13_Sub-Sub/ITF_SubsystemTransport.TcIO
INTERFACE ITF_SubsystemTransport EXTENDS __System.IQueryInterface

METHOD M_CallInterface : BOOL
VAR_IN_OUT
	mErrorData				: ST_ErrorDataSet; // Error data
END_VAR
END_METHOD

METHOD M_GetTransportData : REFERENCE TO ST_TransportData
END_METHOD

METHOD M_Init : BOOL
VAR_INPUT
	mInit			: BOOL; // Force init
END_VAR
END_METHOD

METHOD M_MoveTU_DataIndex : DINT
END_METHOD

END_INTERFACE

// ---- 20_Product/10_BCF/11_Conv/11_Com/13_Sub-Sub/ITF_SubsystemTransportEmulation.TcIO
INTERFACE ITF_SubsystemTransportEmulation EXTENDS __System.IQueryInterface

METHOD M_CallInterface : BOOL
END_METHOD

METHOD M_GetTransportData : REFERENCE TO ST_TransportDataEmulation
END_METHOD

METHOD M_Init : BOOL
VAR_INPUT
	mInit			: BOOL; // Force init
END_VAR
END_METHOD

METHOD M_MoveTU_DataIndex : DINT
END_METHOD

END_INTERFACE

// ---- 20_Product/30_Toolbox/16_Sequencing/02_ITFs/I_BranchCheckpoint.TcIO
/// Branch interface 
INTERFACE I_BranchCheckpoint

/// Searches if a checkpoint can be found on a specific branch
/// Returns true if found, false = not found 
METHOD M_IsOnBranches : BOOL
VAR_INPUT
	mRecursive	: BOOL := FALSE; // Search recursive through the whole tree
END_VAR
VAR_IN_OUT CONSTANT
	mCheckpointID	: STRING(5); // Last checkpoint id	
END_VAR
END_METHOD

/// Identifier for checkpoint
{attribute 'monitoring' := 'call'}
{attribute 'suppress_wrn_C0410'}
PROPERTY P_CheckpointID : REFERENCE TO STRING(5)
GET
END_GET
END_PROPERTY

END_INTERFACE

// ---- 20_Product/30_Toolbox/16_Sequencing/02_ITFs/I_SeqEstimateNext.TcIO
/// Sequencing estimate next interface
INTERFACE I_SeqEstimateNext

/// Checks if requesting TU is next in sequence
METHOD M_IsNextInSequence : BOOL // True = Next in Sequence, otherwise FALSE
VAR_INPUT
	mTU_Index			: DINT; // Requesting TU Index
END_VAR
VAR_IN_OUT
	mTU_Data			: ST_TU_Data; // Tu Data
END_VAR
END_METHOD

END_INTERFACE

// ---- 20_Product/30_Toolbox/17_WindowTracking/10_Core/02_ITFs/I_Encoder.TcIO
/// Provide access to encoder data
INTERFACE I_Encoder EXTENDS __System.IQueryInterface

/// Encoder data
{attribute 'suppress_wrn_C0410'}
PROPERTY P_EncoderData : REFERENCE TO ST_EncoderData
GET
END_GET
END_PROPERTY

END_INTERFACE

// ---- 20_Product/30_Toolbox/17_WindowTracking/10_Core/02_ITFs/I_TrackingActionListener.TcIO
/// Window Tracking action
INTERFACE I_TrackingActionListener EXTENDS __System.IQueryInterface

METHOD M_ActionZoneChangedEvent
VAR_INPUT
	mZoneIndex	: UINT; // Deleted zone index
	mZoneData	: ST_WindowTrackingZone; // Data of deleted zone
END_VAR
END_METHOD

/// Zone deleted
METHOD M_ActionZoneDeletedEvent
VAR_INPUT
	mZoneIndex	: UINT; // Deleted zone index
	mZoneData	: ST_WindowTrackingZone; // Data of deleted zone
END_VAR
END_METHOD

END_INTERFACE

// ---- 20_Product/30_Toolbox/17_WindowTracking/10_Core/02_ITFs/I_TrackingMaster.TcIO
/// TrackingMaster - Allows access to WindowTracking
INTERFACE I_TrackingMaster EXTENDS __SYSTEM.IQueryInterface

/// Tracking is ready for interactions (e.g. Conveyor is on constant speed)
PROPERTY P_TrackingReady : BOOL
GET
END_GET
END_PROPERTY

PROPERTY P_WindowTracking : I_WindowTracking
GET
END_GET
END_PROPERTY

END_INTERFACE

// ---- 20_Product/30_Toolbox/17_WindowTracking/10_Core/02_ITFs/I_WindowTracking.TcIO
/// Implements window tracking funcitonality
INTERFACE I_WindowTracking EXTENDS __System.IQueryInterface

/// Adds a TU to the beginning of the zone
METHOD M_AddTU : BOOL // Returns true successfully, otherwise false (Zone not found, Zone to small or already occupied)
VAR_INPUT
	mZoneIndex				: UINT;	// Zone index 
	mTU_Index				: DINT; // Index of TU to add
	mLength					: UINT; // Length of TU to be added [mm]
	mTU_Offset				: UINT; // Relative TU offset position in zone [mm]
END_VAR
END_METHOD

/// Adds a TU to the tracking by creating a Zone and setting the front edge.
/// The add process is completed by triggering M_AddTU_RearEdge
METHOD M_AddTU_FE : UINT // Returns ZoneIndex > 0 if successfully, otherwise 0
VAR_INPUT
	mTU_Index			: DINT; // Index of TU to add
	mAbsolutePosition	: UDINT; // Position where a TU should be added
	miActionListener	: I_TrackingActionListener; // Action listener of the created zone
END_VAR
END_METHOD

/// Completes an AddTU process which was initiated by M_AddTU_FrontEdge
METHOD M_AddTU_RE : UINT // Returns ZoneIndex > 0 if successfully, otherwise 0
VAR_INPUT
	mAbsolutePosition		: UDINT; // Position where a TU should be added
	mZoneIndex				: UINT;	// Zone index to be completed
END_VAR
END_METHOD

/// Allocates a fixed zone (Can not be shifted)
/// at a specific position. Position needs to be free. 
METHOD M_AllocateFixedZone : UINT; // > 0 Allocated successfully, otherwise 0
VAR_INPUT
	mActionId				: INT; (* ID of action requests zone - 
								     (0 = Only allocation, but free to be used by other acitons) *)
	mAbsolutePosition		: UDINT; // Absolute position on tracking [mm]
	mLength					: UINT; // Length of Zone to be allocated [mm]
	miActionListener		: I_TrackingActionListener; // Action listener of the created zone
	mPositionToLive			: UDINT; // Period of validity until allocation gets deleted automatically (0 = disabled)
END_VAR
END_METHOD

/// Looks from position ascending for enough space to allocate a new Zone.
METHOD M_AllocateNextFreeZone : UINT; // >0 Index of allocated zone, otherwise 0
VAR_INPUT
	mActionId				: INT; (* ID of action which requests zone - 
								     (0 = Only allocation, but free to be used by other actions) *)
	mAbsolutePosition		: UDINT; // Absolute position on tracking [mm]
	mLength					: UINT; // Length of Zone to be allocated [mm]
	mMaxDistance			: UDINT; (* Max distance in which begin of a zone is allowed to be allocated (0=Complete distance) 
										Remark: Multiple of windowsize *)
	miActionListener		: I_TrackingActionListener; // Action listener of the created zone
	mPositionToLive			: UDINT; // Absolute position until allocation gets deleted automatically if not used (0 = disabled)
END_VAR
END_METHOD

// Assigns an already allocated but free zone, beginning at absolute position upstream
// Remark: No zones are allocated, only existing zones are considered.
METHOD M_AssignNextFreeZone : UINT // Returns index of assigned zone if successful, otherwise 0
VAR_INPUT
	mActionId				: INT; // ID of action which requests zone (<>0)
	mAbsolutePosition		: UDINT; // Absolute Start position on the tracking [mm]
	mMaxDistance			: UDINT; // Max distance in which begin of a zone is allowed to be for assignment (0=Complete distance) 
	mLength					: UINT; // Length of Zone to be allocated [mm]
	miActionListener		: I_TrackingActionListener; // Action listener of the created zone
	mPositionToLive			: UDINT; // Absolute position until allocation gets deleted automatically if not used (0 = disabled)
END_VAR
END_METHOD

/// Delete a zone and all related windows
/// Remark: Including zones with physical TUs 
METHOD M_DeleteZone : BOOL // Returns true if successful, otherwise false
VAR_INPUT
	mZoneIndex 				: UINT; // Zone index to delete
END_VAR
END_METHOD

/// Enlarges a zone by given value to upstream direction
METHOD M_EnlargeZone : BOOL
VAR_INPUT
	mZoneIndex 				: UINT; // Zone index to enlarge
	mAdditionalLength		: UINT; // Add this length to existing zone [mm]
	mShiftFrontEdge			: BOOL; // Shift front edge for reduction
END_VAR
END_METHOD

/// Marks all windows and zones in an area to be flushed.
/// (e.g. because of an error the TU position is not reliable anymore)
/// Remark: This includes empty windows as well
METHOD M_FlushDistance : BOOL // Returns true if successful, otherwise false
VAR_INPUT
	mAbsoluteStartPosition		: UDINT; // Position to start marking [mm]
	mAbsoluteEndPosition		: UDINT; // Position to stop marking [mm]
END_VAR
END_METHOD

/// Converts a tracking position into the absolute position regarding tracking length
METHOD M_GetAbsolutePosition : UDINT // Absolute position releated to Tracking length [mm]
VAR_INPUT
	mTrackingPosition			: UDINT; // Tracking position on tracking 
END_VAR
END_METHOD

/// Returns distance to end of tu from observation point. 
/// Position 0 = observation point, Position Max = Observation point plus half tracking length.
/// Remark: In order to reduce the area use M_IsZoneInRange.
METHOD M_GetDistanceToTU_End : DINT // Returns distance to tu end. x < 0 Zone has already passed by x
VAR_INPUT
	mAbsolutePosition		: UDINT; // Absolute position to watch
	mZoneIndex				: UINT; // Index to be measured
END_VAR
END_METHOD

/// Returns distance to begin of TU in Zone from observation point.
/// Remark: Positions after Tracking length are counter as in front of observation point
METHOD M_GetDistanceToTU_Start : DINT // Returns distance to zone start. x < 0 Zone has already passed by x
VAR_INPUT
	mAbsolutePosition		: UDINT; // Absolute position to watch
	mZoneIndex				: UINT; // Index to be measured
END_VAR
END_METHOD

/// Returns distance to end of zone from observation point. 
/// Position 0 = observation point, Position Max = Observation point plus half tracking length.
/// Remark: In order to reduce the area use M_IsZoneInRange.
METHOD M_GetDistanceToZoneEnd : DINT // Returns distance to zone end. x < 0 Zone has already passed by x
VAR_INPUT
	mAbsolutePosition		: UDINT; // Absolute position to watch
	mZoneIndex				: UINT; // Index to be measured
END_VAR
END_METHOD

/// Returns distance to begin of zone from observation point.
/// Remark: Positions after Tracking length are counter as in front of observation point
METHOD M_GetDistanceToZoneStart : DINT // Returns distance to zone start. x < 0 Zone has already passed by x
VAR_INPUT
	mAbsolutePosition		: UDINT; // Absolute position to watch
	mZoneIndex				: UINT; // Index to be measured
END_VAR
END_METHOD

/// Returns first zone index that can be found between start and end position
METHOD M_GetFirstZoneIndex : UINT // Returns ZoneIndex > 0, otherwise 0
VAR_INPUT
	mAbsoluteStartPosition	: UDINT; // Start position on the tracking [mm]
	mAbsoluteEndPosition	: UDINT; // End position on the tracking [mm]
	mOnlyZonesWithTU		: BOOL; // Check only zones with physical TU
END_VAR
END_METHOD

